LIN {X 0,Y 418.244,Z 286.013,A -85,B 0,C 180,E1 -10136.324,E2 -10136.324} C_VEL
LIN {X 0,Y 418.278,Z 286.189,A -85,B 0,C 180,E1 -10136.962,E2 -10136.962} C_VEL
LIN {X 0,Y 422.235,Z 301.677,A -85,B 0,C 180,E1 -10140.044,E2 -10140.044} C_VEL
LIN {X 0,Y 424.407,Z 311.611,A -85,B 0,C 180,E1 -10141.923,E2 -10141.923} C_VEL
LIN {X 0,Y 424.445,Z 314.254,A -85,B 0,C 180,E1 -10142.379,E2 -10142.379} C_VEL
LIN {X 0,Y 424.103,Z 317.879,A -85,B 0,C 180,E1 -10142.98,E2 -10142.98} C_VEL
LIN {X 0,Y 430.223,Z 348.762,A -85,B 0,C 180,E1 -10143.957,E2 -10143.957} C_VEL
LIN {X 0,Y 430.634,Z 351.197,A -85,B 0,C 180,E1 -10144.027,E2 -10144.027} C_VEL
LIN {X 0,Y 428.256,Z 483.679,A -85,B 0,C 180,E1 -10146.294,E2 -10146.294} C_VEL
LIN {X 0,Y 427.572,Z 499.207,A -85,B 0,C 180,E1 -10146.735,E2 -10146.735} C_VEL
LIN {X 0,Y 426.692,Z 513.897,A -85,B 0,C 180,E1 -10147.343,E2 -10147.343} C_VEL
LIN {X 0,Y 425.714,Z 527.179,A -85,B 0,C 180,E1 -10148.068,E2 -10148.068} C_VEL
LIN {X 0,Y 424.501,Z 541.084,A -85,B 0,C 180,E1 -10149.022,E2 -10149.022} C_VEL
LIN {X 0,Y 423.263,Z 553.827,A -85,B 0,C 180,E1 -10150.1,E2 -10150.1} C_VEL
LIN {X 0,Y 421.996,Z 566.72,A -85,B 0,C 180,E1 -10151.428,E2 -10151.428} C_VEL
LIN {X 0,Y 420.886,Z 577.517,A -85,B 0,C 180,E1 -10152.76,E2 -10152.76} C_VEL
LIN {X 0,Y 419.829,Z 587.51,A -85,B 0,C 180,E1 -10154.216,E2 -10154.216} C_VEL
LIN {X 0,Y 418.872,Z 597.29,A -85,B 0,C 180,E1 -10155.92,E2 -10155.92} C_VEL
LIN {X 0,Y 418.217,Z 605.457,A -85,B 0,C 180,E1 -10157.628,E2 -10157.628} C_VEL
LIN {X 0,Y 417.695,Z 612.208,A -85,B 0,C 180,E1 -10159.334,E2 -10159.334} C_VEL
LIN {X 0,Y 417.31,Z 618.446,A -85,B 0,C 180,E1 -10161.282,E2 -10161.282} C_VEL
LIN {X 0,Y 417.147,Z 623.274,A -85,B 0,C 180,E1 -10163.227,E2 -10163.227} C_VEL
LIN {X 0,Y 417.046,Z 626.811,A -85,B 0,C 180,E1 -10165.167,E2 -10165.167} C_VEL
LIN {X 0,Y 417.01,Z 629.139,A -85,B 0,C 180,E1 -10167.102,E2 -10167.102} C_VEL
LIN {X 0,Y 417.008,Z 630.31,A -85,B 0,C 180,E1 -10169.034,E2 -10169.034} C_VEL
LIN {X 0,Y 417.008,Z 630.308,A -85,B 0,C 180,E1 -10170.966,E2 -10170.966} C_VEL
LIN {X 0,Y 417.01,Z 629.131,A -85,B 0,C 180,E1 -10172.898,E2 -10172.898} C_VEL
LIN {X 0,Y 417.025,Z 626.8,A -85,B 0,C 180,E1 -10174.834,E2 -10174.834} C_VEL
LIN {X 0,Y 417.139,Z 623.267,A -85,B 0,C 180,E1 -10176.773,E2 -10176.773} C_VEL
LIN {X 0,Y 417.31,Z 618.438,A -85,B 0,C 180,E1 -10178.718,E2 -10178.718} C_VEL
LIN {X 0,Y 417.694,Z 612.188,A -85,B 0,C 180,E1 -10180.666,E2 -10180.666} C_VEL
LIN {X 0,Y 418.223,Z 605.432,A -85,B 0,C 180,E1 -10182.372,E2 -10182.372} C_VEL
LIN {X 0,Y 419.012,Z 596.002,A -85,B 0,C 180,E1 -10184.323,E2 -10184.323} C_VEL
LIN {X 0,Y 419.969,Z 585.957,A -85,B 0,C 180,E1 -10186.028,E2 -10186.028} C_VEL
LIN {X 0,Y 421.237,Z 574.541,A -85,B 0,C 180,E1 -10187.629,E2 -10187.629} C_VEL
LIN {X 0,Y 422.391,Z 562.305,A -85,B 0,C 180,E1 -10189.058,E2 -10189.058} C_VEL
LIN {X 0,Y 423.709,Z 549.847,A -85,B 0,C 180,E1 -10190.258,E2 -10190.258} C_VEL
LIN {X 0,Y 424.949,Z 536.202,A -85,B 0,C 180,E1 -10191.336,E2 -10191.336} C_VEL
LIN {X 0,Y 426.1,Z 522.072,A -85,B 0,C 180,E1 -10192.229,E2 -10192.229} C_VEL
LIN {X 0,Y 427.157,Z 506.655,A -85,B 0,C 180,E1 -10192.975,E2 -10192.975} C_VEL
LIN {X 0,Y 427.948,Z 491.612,A -85,B 0,C 180,E1 -10193.5,E2 -10193.5} C_VEL
LIN {X 0,Y 428.422,Z 475.672,A -85,B 0,C 180,E1 -10193.857,E2 -10193.857} C_VEL
LIN {X 0,Y 430.58,Z 352.154,A -85,B 0,C 180,E1 -10195.952,E2 -10195.952} C_VEL
LIN {X 0,Y 429.942,Z 347.275,A -85,B 0,C 180,E1 -10196.081,E2 -10196.081} C_VEL
LIN {X 0,Y 424.097,Z 317.761,A -85,B 0,C 180,E1 -10197.032,E2 -10197.032} C_VEL
LIN {X 0,Y 424.547,Z 312.878,A -85,B 0,C 180,E1 -10197.841,E2 -10197.841} C_VEL
LIN {X 0,Y 422.7,Z 303.593,A -85,B 0,C 180,E1 -10199.576,E2 -10199.576} C_VEL
LIN {X 0,Y 419.42,Z 290.486,A -85,B 0,C 180,E1 -10202.152,E2 -10202.152} C_VEL
LIN {X 0,Y 418.237,Z 286.011,A -85,B 0,C 180,E1 -10203.1,E2 -10203.1} C_VEL
LIN {X 0,Y 418.236,Z 286.014,A -85,B 0,C 180,E1 -10206.236,E2 -10206.236} C_VEL
LIN {X 0,Y 418.192,Z 286.02,A -85,B 0,C 180,E1 -10209.687,E2 -10209.687} C_VEL
LIN {X 0,Y 418.202,Z 286.02,A -85,B 0,C 180,E1 -10212.317,E2 -10212.317} C_VEL
LIN {X 0,Y 418.227,Z 286.013,A -85,B 0,C 180,E1 -10215.108,E2 -10215.108} C_VEL
LIN {X 0,Y 418.215,Z 286.016,A -85,B 0,C 180,E1 -10217.764,E2 -10217.764} C_VEL
LIN {X 0,Y 418.225,Z 286.015,A -85,B 0,C 180,E1 -10221.555,E2 -10221.555} C_VEL
LIN {X 0,Y 418.24,Z 286.008,A -85,B 0,C 180,E1 -10225.157,E2 -10225.157} C_VEL
LIN {X 0,Y 418.233,Z 286.01,A -85,B 0,C 180,E1 -10227.471,E2 -10227.471} C_VEL
LIN {X 0,Y 418.252,Z 286.007,A -85,B 0,C 180,E1 -10230.897,E2 -10230.897} C_VEL
LIN {X 0,Y 418.207,Z 286.017,A -85,B 0,C 180,E1 -10234.092,E2 -10234.092} C_VEL
LIN {X 0,Y 418.216,Z 286.014,A -85,B 0,C 180,E1 -10237.263,E2 -10237.263} C_VEL
LIN {X 0,Y 418.272,Z 285.991,A -85,B 0,C 180,E1 -10240.364,E2 -10240.364} C_VEL
LIN {X 0,Y 418.304,Z 286,A -85,B 0,C 180,E1 -10243.404,E2 -10243.404} C_VEL
LIN {X 0,Y 418.334,Z 285.993,A -85,B 0,C 180,E1 -10247,E2 -10247} C_VEL
LIN {X 0,Y 418.306,Z 285.996,A -85,B 0,C 180,E1 -10250.328,E2 -10250.328} C_VEL
LIN {X 0,Y 418.448,Z 285.988,A -85,B 0,C 180,E1 -10253.248,E2 -10253.248} C_VEL
LIN {X 0,Y 418.307,Z 285.999,A -85,B 0,C 180,E1 -10255.181,E2 -10255.181} C_VEL
LIN {X 0,Y 418.52,Z 285.97,A -85,B 0,C 180,E1 -10258.075,E2 -10258.075} C_VEL
LIN {X 0,Y 418.394,Z 285.993,A -85,B 0,C 180,E1 -10260.963,E2 -10260.963} C_VEL
LIN {X 0,Y 418.469,Z 285.978,A -85,B 0,C 180,E1 -10262.888,E2 -10262.888} C_VEL
LIN {X 0,Y 418.452,Z 285.98,A -85,B 0,C 180,E1 -10266.593,E2 -10266.593} C_VEL
LIN {X 0,Y 418.324,Z 285.999,A -85,B 0,C 180,E1 -10269.672,E2 -10269.672} C_VEL
LIN {X 0,Y 418.335,Z 286.002,A -85,B 0,C 180,E1 -10273.001,E2 -10273.001} C_VEL
LIN {X 0,Y 418.301,Z 286.004,A -85,B 0,C 180,E1 -10276.735,E2 -10276.735} C_VEL
LIN {X 0,Y 418.259,Z 285.992,A -85,B 0,C 180,E1 -10279.79,E2 -10279.79} C_VEL
LIN {X 0,Y 418.227,Z 286.008,A -85,B 0,C 180,E1 -10282.737,E2 -10282.737} C_VEL
LIN {X 0,Y 418.251,Z 286.002,A -85,B 0,C 180,E1 -10285.905,E2 -10285.905} C_VEL
LIN {X 0,Y 418.26,Z 286.005,A -85,B 0,C 180,E1 -10289.105,E2 -10289.105} C_VEL
LIN {X 0,Y 418.234,Z 286.009,A -85,B 0,C 180,E1 -10292.529,E2 -10292.529} C_VEL
LIN {X 0,Y 418.234,Z 286.01,A -85,B 0,C 180,E1 -10296.025,E2 -10296.025} C_VEL
LIN {X 0,Y 418.238,Z 286.007,A -85,B 0,C 180,E1 -10299.684,E2 -10299.684} C_VEL
LIN {X 0,Y 418.223,Z 286.013,A -85,B 0,C 180,E1 -10302.322,E2 -10302.322} C_VEL
LIN {X 0,Y 418.23,Z 286.015,A -85,B 0,C 180,E1 -10305.11,E2 -10305.11} C_VEL
LIN {X 0,Y 418.235,Z 286.012,A -85,B 0,C 180,E1 -10307.768,E2 -10307.768} C_VEL
LIN {X 0,Y 418.254,Z 286.007,A -85,B 0,C 180,E1 -10310.619,E2 -10310.619} C_VEL
LIN {X 0,Y 418.239,Z 286.008,A -85,B 0,C 180,E1 -10313.977,E2 -10313.977} C_VEL
LIN {X 0,Y 418.254,Z 286.009,A -85,B 0,C 180,E1 -10317.157,E2 -10317.157} C_VEL
LIN {X 0,Y 418.268,Z 286.038,A -85,B 0,C 180,E1 -10320.426,E2 -10320.426} C_VEL
LIN {X 0,Y 421.092,Z 297.257,A -85,B 0,C 180,E1 -10322.844,E2 -10322.844} C_VEL
LIN {X 0,Y 429.309,Z 316.827,A -85,B 0,C 180,E1 -10323.769,E2 -10323.769} C_VEL
LIN {X 0,Y 430.945,Z 324.515,A -85,B 0,C 180,E1 -10324.017,E2 -10324.017} C_VEL
LIN {X 0,Y 428.589,Z 458.839,A -85,B 0,C 180,E1 -10326.313,E2 -10326.313} C_VEL
LIN {X 0,Y 428.076,Z 473.456,A -85,B 0,C 180,E1 -10326.7,E2 -10326.7} C_VEL
LIN {X 0,Y 427.345,Z 488.698,A -85,B 0,C 180,E1 -10327.299,E2 -10327.299} C_VEL
LIN {X 0,Y 426.339,Z 503.778,A -85,B 0,C 180,E1 -10328.102,E2 -10328.102} C_VEL
LIN {X 0,Y 425.211,Z 517.76,A -85,B 0,C 180,E1 -10329.059,E2 -10329.059} C_VEL
LIN {X 0,Y 423.983,Z 530.538,A -85,B 0,C 180,E1 -10330.135,E2 -10330.135} C_VEL
LIN {X 0,Y 422.724,Z 543.427,A -85,B 0,C 180,E1 -10331.464,E2 -10331.464} C_VEL
LIN {X 0,Y 421.603,Z 554.154,A -85,B 0,C 180,E1 -10332.79,E2 -10332.79} C_VEL
LIN {X 0,Y 421.269,Z 557.507,A -85,B 0,C 180,E1 -10333.249,E2 -10333.249} C_VEL
LIN {X 0,Y 420.236,Z 561.612,A -85,B 0,C 180,E1 -10333.811,E2 -10333.811} C_VEL
LIN {X 0,Y 416.771,Z 568.053,A -85,B 0,C 180,E1 -10334.729,E2 -10334.729} C_VEL
LIN {X 0,Y 413.273,Z 574.004,A -85,B 0,C 180,E1 -10335.715,E2 -10335.715} C_VEL
LIN {X 0,Y 412.208,Z 577.344,A -85,B 0,C 180,E1 -10336.377,E2 -10336.377} C_VEL
LIN {X 0,Y 411.56,Z 585.076,A -85,B 0,C 180,E1 -10338.176,E2 -10338.176} C_VEL
LIN {X 0,Y 410.84,Z 592.015,A -85,B 0,C 180,E1 -10340.151,E2 -10340.151} C_VEL
LIN {X 0,Y 410.445,Z 597.464,A -85,B 0,C 180,E1 -10342.127,E2 -10342.127} C_VEL
LIN {X 0,Y 410.194,Z 601.578,A -85,B 0,C 180,E1 -10344.1,E2 -10344.1} C_VEL
LIN {X 0,Y 409.99,Z 604.471,A -85,B 0,C 180,E1 -10346.068,E2 -10346.068} C_VEL
LIN {X 0,Y 410.008,Z 606.209,A -85,B 0,C 180,E1 -10348.035,E2 -10348.035} C_VEL
LIN {X 0,Y 409.925,Z 606.819,A -85,B 0,C 180,E1 -10350,E2 -10350} C_VEL
LIN {X 0,Y 410.008,Z 606.257,A -85,B 0,C 180,E1 -10351.965,E2 -10351.965} C_VEL
LIN {X 0,Y 409.98,Z 604.584,A -85,B 0,C 180,E1 -10353.932,E2 -10353.932} C_VEL
LIN {X 0,Y 410.182,Z 601.751,A -85,B 0,C 180,E1 -10355.9,E2 -10355.9} C_VEL
LIN {X 0,Y 410.411,Z 597.698,A -85,B 0,C 180,E1 -10357.874,E2 -10357.874} C_VEL
LIN {X 0,Y 410.824,Z 592.321,A -85,B 0,C 180,E1 -10359.85,E2 -10359.85} C_VEL
LIN {X 0,Y 411.541,Z 585.465,A -85,B 0,C 180,E1 -10361.825,E2 -10361.825} C_VEL
LIN {X 0,Y 412.292,Z 576.91,A -85,B 0,C 180,E1 -10363.806,E2 -10363.806} C_VEL
LIN {X 0,Y 413.318,Z 567.808,A -85,B 0,C 180,E1 -10365.534,E2 -10365.534} C_VEL
LIN {X 0,Y 414.347,Z 558.53,A -85,B 0,C 180,E1 -10367.012,E2 -10367.012} C_VEL
LIN {X 0,Y 415.663,Z 546.61,A -85,B 0,C 180,E1 -10368.6,E2 -10368.6} C_VEL
LIN {X 0,Y 416.981,Z 534.265,A -85,B 0,C 180,E1 -10369.956,E2 -10369.956} C_VEL
LIN {X 0,Y 418.37,Z 520.731,A -85,B 0,C 180,E1 -10371.171,E2 -10371.171} C_VEL
LIN {X 0,Y 419.534,Z 507.419,A -85,B 0,C 180,E1 -10372.142,E2 -10372.142} C_VEL
LIN {X 0,Y 420.633,Z 492.721,A -85,B 0,C 180,E1 -10372.988,E2 -10372.988} C_VEL
LIN {X 0,Y 421.422,Z 478.095,A -85,B 0,C 180,E1 -10373.625,E2 -10373.625} C_VEL
LIN {X 0,Y 422.01,Z 463.194,A -85,B 0,C 180,E1 -10374.079,E2 -10374.079} C_VEL
LIN {X 0,Y 422.988,Z 418.773,A -85,B 0,C 180,E1 -10374.87,E2 -10374.87} C_VEL
LIN {X 0,Y 424.551,Z 324.982,A -85,B 0,C 180,E1 -10376.498,E2 -10376.498} C_VEL
LIN {X 0,Y 422.627,Z 317.569,A -85,B 0,C 180,E1 -10376.767,E2 -10376.767} C_VEL
LIN {X 0,Y 413.797,Z 297.173,A -85,B 0,C 180,E1 -10377.792,E2 -10377.792} C_VEL
LIN {X 0,Y 411.215,Z 286.891,A -85,B 0,C 180,E1 -10380.134,E2 -10380.134} C_VEL
LIN {X 0,Y 411.204,Z 286.894,A -85,B 0,C 180,E1 -10383.155,E2 -10383.155} C_VEL
LIN {X 0,Y 411.191,Z 286.894,A -85,B 0,C 180,E1 -10386.552,E2 -10386.552} C_VEL
LIN {X 0,Y 411.208,Z 286.884,A -85,B 0,C 180,E1 -10389.727,E2 -10389.727} C_VEL
LIN {X 0,Y 411.168,Z 286.894,A -85,B 0,C 180,E1 -10393.133,E2 -10393.133} C_VEL
LIN {X 0,Y 411.161,Z 286.893,A -85,B 0,C 180,E1 -10395.88,E2 -10395.88} C_VEL
LIN {X 0,Y 411.154,Z 286.882,A -85,B 0,C 180,E1 -10398.771,E2 -10398.771} C_VEL
LIN {X 0,Y 411.182,Z 286.884,A -85,B 0,C 180,E1 -10402.025,E2 -10402.025} C_VEL
LIN {X 0,Y 411.185,Z 286.891,A -85,B 0,C 180,E1 -10405.664,E2 -10405.664} C_VEL
LIN {X 0,Y 411.18,Z 286.875,A -85,B 0,C 180,E1 -10409.151,E2 -10409.151} C_VEL
LIN {X 0,Y 411.258,Z 286.882,A -85,B 0,C 180,E1 -10412.698,E2 -10412.698} C_VEL
LIN {X 0,Y 411.201,Z 286.887,A -85,B 0,C 180,E1 -10415.783,E2 -10415.783} C_VEL
LIN {X 0,Y 411.186,Z 286.889,A -85,B 0,C 180,E1 -10418.965,E2 -10418.965} C_VEL
LIN {X 0,Y 411.234,Z 286.878,A -85,B 0,C 180,E1 -10422.084,E2 -10422.084} C_VEL
LIN {X 0,Y 411.247,Z 286.882,A -85,B 0,C 180,E1 -10425.147,E2 -10425.147} C_VEL
LIN {X 0,Y 411.27,Z 286.877,A -85,B 0,C 180,E1 -10428.167,E2 -10428.167} C_VEL
LIN {X 0,Y 411.427,Z 286.856,A -85,B 0,C 180,E1 -10432.191,E2 -10432.191} C_VEL
LIN {X 0,Y 411.432,Z 286.858,A -85,B 0,C 180,E1 -10434.117,E2 -10434.117} C_VEL
LIN {X 0,Y 411.497,Z 286.85,A -85,B 0,C 180,E1 -10438.042,E2 -10438.042} C_VEL
LIN {X 0,Y 411.622,Z 286.83,A -85,B 0,C 180,E1 -10440,E2 -10440} C_VEL
LIN {X 0,Y 411.421,Z 286.86,A -85,B 0,C 180,E1 -10442.937,E2 -10442.937} C_VEL
LIN {X 0,Y 411.419,Z 286.863,A -85,B 0,C 180,E1 -10446.868,E2 -10446.868} C_VEL
LIN {X 0,Y 411.27,Z 286.874,A -85,B 0,C 180,E1 -10449.839,E2 -10449.839} C_VEL
LIN {X 0,Y 411.294,Z 286.87,A -85,B 0,C 180,E1 -10453.104,E2 -10453.104} C_VEL
LIN {X 0,Y 411.247,Z 286.88,A -85,B 0,C 180,E1 -10456.889,E2 -10456.889} C_VEL
LIN {X 0,Y 411.22,Z 286.888,A -85,B 0,C 180,E1 -10459.987,E2 -10459.987} C_VEL
LIN {X 0,Y 411.176,Z 286.891,A -85,B 0,C 180,E1 -10463.149,E2 -10463.149} C_VEL
LIN {X 0,Y 411.164,Z 286.892,A -85,B 0,C 180,E1 -10466.386,E2 -10466.386} C_VEL
LIN {X 0,Y 411.188,Z 286.89,A -85,B 0,C 180,E1 -10469.714,E2 -10469.714} C_VEL
LIN {X 0,Y 411.195,Z 286.882,A -85,B 0,C 180,E1 -10473.157,E2 -10473.157} C_VEL
LIN {X 0,Y 411.179,Z 286.889,A -85,B 0,C 180,E1 -10476.552,E2 -10476.552} C_VEL
LIN {X 0,Y 411.159,Z 286.884,A -85,B 0,C 180,E1 -10479.721,E2 -10479.721} C_VEL
LIN {X 0,Y 411.157,Z 286.893,A -85,B 0,C 180,E1 -10483.136,E2 -10483.136} C_VEL
LIN {X 0,Y 411.156,Z 286.896,A -85,B 0,C 180,E1 -10485.883,E2 -10485.883} C_VEL
LIN {X 0,Y 411.14,Z 286.895,A -85,B 0,C 180,E1 -10488.775,E2 -10488.775} C_VEL
LIN {X 0,Y 411.176,Z 286.892,A -85,B 0,C 180,E1 -10492.026,E2 -10492.026} C_VEL
LIN {X 0,Y 411.201,Z 286.89,A -85,B 0,C 180,E1 -10495.667,E2 -10495.667} C_VEL
LIN {X 0,Y 411.228,Z 287.031,A -85,B 0,C 180,E1 -10496.518,E2 -10496.518} C_VEL
LIN {X 0,Y 415.224,Z 302.546,A -85,B 0,C 180,E1 -10499.679,E2 -10499.679} C_VEL
LIN {X 0,Y 417.696,Z 314.046,A -85,B 0,C 180,E1 -10501.894,E2 -10501.894} C_VEL
LIN {X 0,Y 417.508,Z 317.887,A -85,B 0,C 180,E1 -10502.524,E2 -10502.524} C_VEL
LIN {X 0,Y 423.554,Z 348.293,A -85,B 0,C 180,E1 -10503.51,E2 -10503.51} C_VEL
LIN {X 0,Y 424.204,Z 351.82,A -85,B 0,C 180,E1 -10503.619,E2 -10503.619} C_VEL
LIN {X 0,Y 421.839,Z 481.988,A -85,B 0,C 180,E1 -10505.878,E2 -10505.878} C_VEL
LIN {X 0,Y 421.199,Z 497.183,A -85,B 0,C 180,E1 -10506.296,E2 -10506.296} C_VEL
LIN {X 0,Y 420.276,Z 511.874,A -85,B 0,C 180,E1 -10506.886,E2 -10506.886} C_VEL
LIN {X 0,Y 419.259,Z 524.987,A -85,B 0,C 180,E1 -10507.583,E2 -10507.583} C_VEL
LIN {X 0,Y 417.986,Z 539.298,A -85,B 0,C 180,E1 -10508.55,E2 -10508.55} C_VEL
LIN {X 0,Y 416.671,Z 552.33,A -85,B 0,C 180,E1 -10509.643,E2 -10509.643} C_VEL
LIN {X 0,Y 415.395,Z 564.368,A -85,B 0,C 180,E1 -10510.865,E2 -10510.865} C_VEL
LIN {X 0,Y 414.275,Z 575.524,A -85,B 0,C 180,E1 -10512.221,E2 -10512.221} C_VEL
LIN {X 0,Y 413.049,Z 585.786,A -85,B 0,C 180,E1 -10513.696,E2 -10513.696} C_VEL
LIN {X 0,Y 412.058,Z 595.825,A -85,B 0,C 180,E1 -10515.43,E2 -10515.43} C_VEL
LIN {X 0,Y 411.262,Z 604.165,A -85,B 0,C 180,E1 -10517.165,E2 -10517.165} C_VEL
LIN {X 0,Y 410.853,Z 610.183,A -85,B 0,C 180,E1 -10518.655,E2 -10518.655} C_VEL
LIN {X 0,Y 410.32,Z 616.806,A -85,B 0,C 180,E1 -10520.636,E2 -10520.636} C_VEL
LIN {X 0,Y 410.107,Z 621.994,A -85,B 0,C 180,E1 -10522.616,E2 -10522.616} C_VEL
LIN {X 0,Y 409.975,Z 624.995,A -85,B 0,C 180,E1 -10524.097,E2 -10524.097} C_VEL
LIN {X 0,Y 409.893,Z 627.918,A -85,B 0,C 180,E1 -10526.067,E2 -10526.067} C_VEL
LIN {X 0,Y 409.961,Z 629.665,A -85,B 0,C 180,E1 -10528.035,E2 -10528.035} C_VEL
LIN {X 0,Y 409.923,Z 630.262,A -85,B 0,C 180,E1 -10530,E2 -10530} C_VEL
LIN {X 0,Y 409.961,Z 629.661,A -85,B 0,C 180,E1 -10531.965,E2 -10531.965} C_VEL
LIN {X 0,Y 409.89,Z 627.908,A -85,B 0,C 180,E1 -10533.933,E2 -10533.933} C_VEL
LIN {X 0,Y 409.975,Z 624.984,A -85,B 0,C 180,E1 -10535.903,E2 -10535.903} C_VEL
LIN {X 0,Y 410.131,Z 620.816,A -85,B 0,C 180,E1 -10537.879,E2 -10537.879} C_VEL
LIN {X 0,Y 410.379,Z 615.293,A -85,B 0,C 180,E1 -10539.861,E2 -10539.861} C_VEL
LIN {X 0,Y 410.991,Z 608.274,A -85,B 0,C 180,E1 -10541.841,E2 -10541.841} C_VEL
LIN {X 0,Y 411.588,Z 600.675,A -85,B 0,C 180,E1 -10543.597,E2 -10543.597} C_VEL
LIN {X 0,Y 412.489,Z 591.709,A -85,B 0,C 180,E1 -10545.312,E2 -10545.312} C_VEL
LIN {X 0,Y 413.472,Z 582.478,A -85,B 0,C 180,E1 -10546.795,E2 -10546.795} C_VEL
LIN {X 0,Y 414.563,Z 572.303,A -85,B 0,C 180,E1 -10548.186,E2 -10548.186} C_VEL
LIN {X 0,Y 415.856,Z 559.74,A -85,B 0,C 180,E1 -10549.626,E2 -10549.626} C_VEL
LIN {X 0,Y 417.28,Z 546.775,A -85,B 0,C 180,E1 -10550.842,E2 -10550.842} C_VEL
LIN {X 0,Y 418.526,Z 534.225,A -85,B 0,C 180,E1 -10551.809,E2 -10551.809} C_VEL
LIN {X 0,Y 419.621,Z 520.739,A -85,B 0,C 180,E1 -10552.656,E2 -10552.656} C_VEL
LIN {X 0,Y 420.639,Z 505.747,A -85,B 0,C 180,E1 -10553.382,E2 -10553.382} C_VEL
LIN {X 0,Y 421.442,Z 491.397,A -85,B 0,C 180,E1 -10553.885,E2 -10553.885} C_VEL
LIN {X 0,Y 421.948,Z 475.45,A -85,B 0,C 180,E1 -10554.247,E2 -10554.247} C_VEL
LIN {X 0,Y 424.196,Z 352.499,A -85,B 0,C 180,E1 -10556.362,E2 -10556.362} C_VEL
LIN {X 0,Y 419.4,Z 326.937,A -85,B 0,C 180,E1 -10557.164,E2 -10557.164} C_VEL
LIN {X 0,Y 417.45,Z 317.556,A -85,B 0,C 180,E1 -10557.497,E2 -10557.497} C_VEL
LIN {X 0,Y 417.685,Z 313.984,A -85,B 0,C 180,E1 -10558.107,E2 -10558.107} C_VEL
LIN {X 0,Y 415.482,Z 303.69,A -85,B 0,C 180,E1 -10560.085,E2 -10560.085} C_VEL
LIN {X 0,Y 412.102,Z 290.329,A -85,B 0,C 180,E1 -10562.782,E2 -10562.782} C_VEL
LIN {X 0,Y 411.21,Z 286.888,A -85,B 0,C 180,E1 -10563.52,E2 -10563.52} C_VEL
LIN {X 0,Y 411.181,Z 286.892,A -85,B 0,C 180,E1 -10566.742,E2 -10566.742} C_VEL
LIN {X 0,Y 411.161,Z 286.895,A -85,B 0,C 180,E1 -10569.719,E2 -10569.719} C_VEL
LIN {X 0,Y 411.156,Z 286.894,A -85,B 0,C 180,E1 -10573.134,E2 -10573.134} C_VEL
LIN {X 0,Y 411.157,Z 286.897,A -85,B 0,C 180,E1 -10575.881,E2 -10575.881} C_VEL
LIN {X 0,Y 411.141,Z 286.895,A -85,B 0,C 180,E1 -10578.773,E2 -10578.773} C_VEL
LIN {X 0,Y 411.172,Z 286.892,A -85,B 0,C 180,E1 -10582.024,E2 -10582.024} C_VEL
LIN {X 0,Y 411.192,Z 286.886,A -85,B 0,C 180,E1 -10585.123,E2 -10585.123} C_VEL
LIN {X 0,Y 411.154,Z 286.896,A -85,B 0,C 180,E1 -10588.002,E2 -10588.002} C_VEL
LIN {X 0,Y 411.169,Z 286.893,A -85,B 0,C 180,E1 -10591.406,E2 -10591.406} C_VEL
LIN {X 0,Y 411.177,Z 286.89,A -85,B 0,C 180,E1 -10594.941,E2 -10594.941} C_VEL
LIN {X 0,Y 411.192,Z 286.89,A -85,B 0,C 180,E1 -10597.913,E2 -10597.913} C_VEL
LIN {X 0,Y 411.206,Z 286.869,A -85,B 0,C 180,E1 -10601.051,E2 -10601.051} C_VEL
LIN {X 0,Y 411.24,Z 286.883,A -85,B 0,C 180,E1 -10604.131,E2 -10604.131} C_VEL
LIN {X 0,Y 411.29,Z 286.866,A -85,B 0,C 180,E1 -10607.165,E2 -10607.165} C_VEL
LIN {X 0,Y 411.26,Z 286.874,A -85,B 0,C 180,E1 -10610.161,E2 -10610.161} C_VEL
LIN {X 0,Y 411.413,Z 286.863,A -85,B 0,C 180,E1 -10613.132,E2 -10613.132} C_VEL
LIN {X 0,Y 411.279,Z 286.874,A -85,B 0,C 180,E1 -10615.099,E2 -10615.099} C_VEL
LIN {X 0,Y 411.49,Z 286.846,A -85,B 0,C 180,E1 -10618.043,E2 -10618.043} C_VEL
LIN {X 0,Y 411.494,Z 286.847,A -85,B 0,C 180,E1 -10621.958,E2 -10621.958} C_VEL
LIN {X 0,Y 411.412,Z 286.857,A -85,B 0,C 180,E1 -10626.596,E2 -10626.596} C_VEL
LIN {X 0,Y 411.306,Z 286.875,A -85,B 0,C 180,E1 -10628.846,E2 -10628.846} C_VEL
LIN {X 0,Y 411.27,Z 286.878,A -85,B 0,C 180,E1 -10631.833,E2 -10631.833} C_VEL
LIN {X 0,Y 411.245,Z 286.881,A -85,B 0,C 180,E1 -10634.853,E2 -10634.853} C_VEL
LIN {X 0,Y 411.234,Z 286.88,A -85,B 0,C 180,E1 -10637.916,E2 -10637.916} C_VEL
LIN {X 0,Y 411.186,Z 286.872,A -85,B 0,C 180,E1 -10641.035,E2 -10641.035} C_VEL
LIN {X 0,Y 411.207,Z 286.886,A -85,B 0,C 180,E1 -10644.217,E2 -10644.217} C_VEL
LIN {X 0,Y 411.25,Z 286.867,A -85,B 0,C 180,E1 -10647.478,E2 -10647.478} C_VEL
LIN {X 0,Y 411.181,Z 286.894,A -85,B 0,C 180,E1 -10650.848,E2 -10650.848} C_VEL
LIN {X 0,Y 411.184,Z 286.889,A -85,B 0,C 180,E1 -10654.336,E2 -10654.336} C_VEL
LIN {X 0,Y 411.185,Z 286.886,A -85,B 0,C 180,E1 -10657.975,E2 -10657.975} C_VEL
LIN {X 0,Y 411.157,Z 286.894,A -85,B 0,C 180,E1 -10661.229,E2 -10661.229} C_VEL
LIN {X 0,Y 411.17,Z 286.893,A -85,B 0,C 180,E1 -10664.491,E2 -10664.491} C_VEL
LIN {X 0,Y 411.173,Z 286.893,A -85,B 0,C 180,E1 -10668.196,E2 -10668.196} C_VEL
LIN {X 0,Y 411.218,Z 286.882,A -85,B 0,C 180,E1 -10670.777,E2 -10670.777} C_VEL
LIN {X 0,Y 411.194,Z 286.885,A -85,B 0,C 180,E1 -10674.472,E2 -10674.472} C_VEL
LIN {X 0,Y 411.205,Z 286.886,A -85,B 0,C 180,E1 -10676.874,E2 -10676.874} C_VEL
LIN {X 0,Y 411.221,Z 286.926,A -85,B 0,C 180,E1 -10680.008,E2 -10680.008} C_VEL
LIN {X 0,Y 413.864,Z 297.254,A -85,B 0,C 180,E1 -10682.324,E2 -10682.324} C_VEL
LIN {X 0,Y 423.139,Z 318.948,A -85,B 0,C 180,E1 -10683.392,E2 -10683.392} C_VEL
LIN {X 0,Y 424.531,Z 325.264,A -85,B 0,C 180,E1 -10683.604,E2 -10683.604} C_VEL
LIN {X 0,Y 422.503,Z 438.469,A -85,B 0,C 180,E1 -10685.559,E2 -10685.559} C_VEL
LIN {X 0,Y 421.964,Z 463.218,A -85,B 0,C 180,E1 -10686.016,E2 -10686.016} C_VEL
LIN {X 0,Y 421.361,Z 478.668,A -85,B 0,C 180,E1 -10686.492,E2 -10686.492} C_VEL
LIN {X 0,Y 420.666,Z 492.476,A -85,B 0,C 180,E1 -10687.098,E2 -10687.098} C_VEL
LIN {X 0,Y 419.612,Z 505.967,A -85,B 0,C 180,E1 -10687.862,E2 -10687.862} C_VEL
LIN {X 0,Y 418.432,Z 519.546,A -85,B 0,C 180,E1 -10688.832,E2 -10688.832} C_VEL
LIN {X 0,Y 417.062,Z 533.318,A -85,B 0,C 180,E1 -10690.048,E2 -10690.048} C_VEL
LIN {X 0,Y 415.783,Z 545.736,A -85,B 0,C 180,E1 -10691.395,E2 -10691.395} C_VEL
LIN {X 0,Y 414.61,Z 556.132,A -85,B 0,C 180,E1 -10692.745,E2 -10692.745} C_VEL
LIN {X 0,Y 413.525,Z 565.772,A -85,B 0,C 180,E1 -10694.222,E2 -10694.222} C_VEL
LIN {X 0,Y 412.462,Z 575.219,A -85,B 0,C 180,E1 -10695.948,E2 -10695.948} C_VEL
LIN {X 0,Y 412.208,Z 577.344,A -85,B 0,C 180,E1 -10696.377,E2 -10696.377} C_VEL
LIN {X 0,Y 411.188,Z 580.565,A -85,B 0,C 180,E1 -10697.056,E2 -10697.056} C_VEL
LIN {X 0,Y 407.883,Z 585.558,A -85,B 0,C 180,E1 -10698.162,E2 -10698.162} C_VEL
LIN {X 0,Y 404.661,Z 590.076,A -85,B 0,C 180,E1 -10699.321,E2 -10699.321} C_VEL
LIN {X 0,Y 403.782,Z 592.508,A -85,B 0,C 180,E1 -10700.074,E2 -10700.074} C_VEL
LIN {X 0,Y 403.391,Z 597.669,A -85,B 0,C 180,E1 -10701.988,E2 -10701.988} C_VEL
LIN {X 0,Y 403.117,Z 601.782,A -85,B 0,C 180,E1 -10703.996,E2 -10703.996} C_VEL
LIN {X 0,Y 402.909,Z 604.675,A -85,B 0,C 180,E1 -10705.999,E2 -10705.999} C_VEL
LIN {X 0,Y 402.921,Z 606.412,A -85,B 0,C 180,E1 -10708.001,E2 -10708.001} C_VEL
LIN {X 0,Y 402.85,Z 607.022,A -85,B 0,C 180,E1 -10710,E2 -10710} C_VEL
LIN {X 0,Y 402.921,Z 606.46,A -85,B 0,C 180,E1 -10711.999,E2 -10711.999} C_VEL
LIN {X 0,Y 402.9,Z 604.786,A -85,B 0,C 180,E1 -10714.001,E2 -10714.001} C_VEL
LIN {X 0,Y 403.106,Z 601.954,A -85,B 0,C 180,E1 -10716.004,E2 -10716.004} C_VEL
LIN {X 0,Y 403.367,Z 597.9,A -85,B 0,C 180,E1 -10718.012,E2 -10718.012} C_VEL
LIN {X 0,Y 403.793,Z 592.524,A -85,B 0,C 180,E1 -10720.023,E2 -10720.023} C_VEL
LIN {X 0,Y 404.558,Z 585.667,A -85,B 0,C 180,E1 -10722.032,E2 -10722.032} C_VEL
LIN {X 0,Y 405.386,Z 577.111,A -85,B 0,C 180,E1 -10724.046,E2 -10724.046} C_VEL
LIN {X 0,Y 406.437,Z 568.01,A -85,B 0,C 180,E1 -10725.803,E2 -10725.803} C_VEL
LIN {X 0,Y 407.535,Z 558.731,A -85,B 0,C 180,E1 -10727.306,E2 -10727.306} C_VEL
LIN {X 0,Y 408.843,Z 547.383,A -85,B 0,C 180,E1 -10728.846,E2 -10728.846} C_VEL
LIN {X 0,Y 410.293,Z 534.464,A -85,B 0,C 180,E1 -10730.295,E2 -10730.295} C_VEL
LIN {X 0,Y 411.752,Z 520.928,A -85,B 0,C 180,E1 -10731.528,E2 -10731.528} C_VEL
LIN {X 0,Y 412.97,Z 507.615,A -85,B 0,C 180,E1 -10732.513,E2 -10732.513} C_VEL
LIN {X 0,Y 414.14,Z 492.366,A -85,B 0,C 180,E1 -10733.399,E2 -10733.399} C_VEL
LIN {X 0,Y 414.975,Z 477.478,A -85,B 0,C 180,E1 -10734.049,E2 -10734.049} C_VEL
LIN {X 0,Y 415.6,Z 462.192,A -85,B 0,C 180,E1 -10734.508,E2 -10734.508} C_VEL
LIN {X 0,Y 417.138,Z 383.214,A -85,B 0,C 180,E1 -10735.912,E2 -10735.912} C_VEL
LIN {X 0,Y 418.166,Z 326.035,A -85,B 0,C 180,E1 -10736.918,E2 -10736.918} C_VEL
LIN {X 0,Y 416.545,Z 320.085,A -85,B 0,C 180,E1 -10737.145,E2 -10737.145} C_VEL
LIN {X 0,Y 407.653,Z 299.871,A -85,B 0,C 180,E1 -10738.189,E2 -10738.189} C_VEL
LIN {X 0,Y 406.567,Z 297.314,A -85,B 0,C 180,E1 -10738.347,E2 -10738.347} C_VEL
LIN {X 0,Y 404.156,Z 287.771,A -85,B 0,C 180,E1 -10740.572,E2 -10740.572} C_VEL
LIN {X 0,Y 404.143,Z 287.772,A -85,B 0,C 180,E1 -10743.811,E2 -10743.811} C_VEL
LIN {X 0,Y 404.135,Z 287.77,A -85,B 0,C 180,E1 -10746.874,E2 -10746.874} C_VEL
LIN {X 0,Y 404.144,Z 287.762,A -85,B 0,C 180,E1 -10750.079,E2 -10750.079} C_VEL
LIN {X 0,Y 404.148,Z 287.769,A -85,B 0,C 180,E1 -10753.083,E2 -10753.083} C_VEL
LIN {X 0,Y 404.142,Z 287.768,A -85,B 0,C 180,E1 -10755.925,E2 -10755.925} C_VEL
LIN {X 0,Y 404.108,Z 287.759,A -85,B 0,C 180,E1 -10758.633,E2 -10758.633} C_VEL
LIN {X 0,Y 404.141,Z 287.765,A -85,B 0,C 180,E1 -10761.492,E2 -10761.492} C_VEL
LIN {X 0,Y 404.166,Z 287.76,A -85,B 0,C 180,E1 -10764.982,E2 -10764.982} C_VEL
LIN {X 0,Y 404.13,Z 287.758,A -85,B 0,C 180,E1 -10768.442,E2 -10768.442} C_VEL
LIN {X 0,Y 404.186,Z 287.76,A -85,B 0,C 180,E1 -10772,E2 -10772} C_VEL
LIN {X 0,Y 404.155,Z 287.767,A -85,B 0,C 180,E1 -10775.333,E2 -10775.333} C_VEL
LIN {X 0,Y 404.128,Z 287.765,A -85,B 0,C 180,E1 -10778.58,E2 -10778.58} C_VEL
LIN {X 0,Y 404.193,Z 287.755,A -85,B 0,C 180,E1 -10781.761,E2 -10781.761} C_VEL
LIN {X 0,Y 404.194,Z 287.764,A -85,B 0,C 180,E1 -10784.881,E2 -10784.881} C_VEL
LIN {X 0,Y 404.243,Z 287.752,A -85,B 0,C 180,E1 -10787.958,E2 -10787.958} C_VEL
LIN {X 0,Y 404.253,Z 287.749,A -85,B 0,C 180,E1 -10790.998,E2 -10790.998} C_VEL
LIN {X 0,Y 404.383,Z 287.736,A -85,B 0,C 180,E1 -10794.014,E2 -10794.014} C_VEL
LIN {X 0,Y 404.466,Z 287.726,A -85,B 0,C 180,E1 -10798.008,E2 -10798.008} C_VEL
LIN {X 0,Y 404.591,Z 287.706,A -85,B 0,C 180,E1 -10800,E2 -10800} C_VEL
LIN {X 0,Y 404.381,Z 287.737,A -85,B 0,C 180,E1 -10802.989,E2 -10802.989} C_VEL
LIN {X 0,Y 404.369,Z 287.74,A -85,B 0,C 180,E1 -10806.988,E2 -10806.988} C_VEL
LIN {X 0,Y 404.234,Z 287.757,A -85,B 0,C 180,E1 -10811.025,E2 -10811.025} C_VEL
LIN {X 0,Y 404.197,Z 287.756,A -85,B 0,C 180,E1 -10814.089,E2 -10814.089} C_VEL
LIN {X 0,Y 404.192,Z 287.757,A -85,B 0,C 180,E1 -10817.193,E2 -10817.193} C_VEL
LIN {X 0,Y 404.153,Z 287.771,A -85,B 0,C 180,E1 -10820.352,E2 -10820.352} C_VEL
LIN {X 0,Y 404.138,Z 287.768,A -85,B 0,C 180,E1 -10823.576,E2 -10823.576} C_VEL
LIN {X 0,Y 404.112,Z 287.771,A -85,B 0,C 180,E1 -10826.883,E2 -10826.883} C_VEL
LIN {X 0,Y 404.135,Z 287.771,A -85,B 0,C 180,E1 -10830.286,E2 -10830.286} C_VEL
LIN {X 0,Y 404.129,Z 287.765,A -85,B 0,C 180,E1 -10833.814,E2 -10833.814} C_VEL
LIN {X 0,Y 404.122,Z 287.768,A -85,B 0,C 180,E1 -10836.874,E2 -10836.874} C_VEL
LIN {X 0,Y 404.109,Z 287.758,A -85,B 0,C 180,E1 -10840.075,E2 -10840.075} C_VEL
LIN {X 0,Y 404.137,Z 287.768,A -85,B 0,C 180,E1 -10843.083,E2 -10843.083} C_VEL
LIN {X 0,Y 404.113,Z 287.773,A -85,B 0,C 180,E1 -10845.923,E2 -10845.923} C_VEL
LIN {X 0,Y 404.095,Z 287.773,A -85,B 0,C 180,E1 -10848.633,E2 -10848.633} C_VEL
LIN {X 0,Y 404.132,Z 287.768,A -85,B 0,C 180,E1 -10851.496,E2 -10851.496} C_VEL
LIN {X 0,Y 404.179,Z 287.765,A -85,B 0,C 180,E1 -10854.984,E2 -10854.984} C_VEL
LIN {X 0,Y 404.185,Z 287.805,A -85,B 0,C 180,E1 -10856.043,E2 -10856.043} C_VEL
LIN {X 0,Y 408.148,Z 303.137,A -85,B 0,C 180,E1 -10859.245,E2 -10859.245} C_VEL
LIN {X 0,Y 410.822,Z 315.386,A -85,B 0,C 180,E1 -10861.659,E2 -10861.659} C_VEL
LIN {X 0,Y 410.869,Z 317.65,A -85,B 0,C 180,E1 -10862.041,E2 -10862.041} C_VEL
LIN {X 0,Y 417.087,Z 348.646,A -85,B 0,C 180,E1 -10863.077,E2 -10863.077} C_VEL
LIN {X 0,Y 417.834,Z 354.261,A -85,B 0,C 180,E1 -10863.234,E2 -10863.234} C_VEL
LIN {X 0,Y 415.365,Z 481.801,A -85,B 0,C 180,E1 -10865.477,E2 -10865.477} C_VEL
LIN {X 0,Y 414.687,Z 496.989,A -85,B 0,C 180,E1 -10865.9,E2 -10865.9} C_VEL
LIN {X 0,Y 413.792,Z 510.383,A -85,B 0,C 180,E1 -10866.437,E2 -10866.437} C_VEL
LIN {X 0,Y 412.683,Z 524.789,A -85,B 0,C 180,E1 -10867.206,E2 -10867.206} C_VEL
LIN {X 0,Y 411.351,Z 539.098,A -85,B 0,C 180,E1 -10868.186,E2 -10868.186} C_VEL
LIN {X 0,Y 409.982,Z 552.129,A -85,B 0,C 180,E1 -10869.295,E2 -10869.295} C_VEL
LIN {X 0,Y 408.504,Z 565.24,A -85,B 0,C 180,E1 -10870.66,E2 -10870.66} C_VEL
LIN {X 0,Y 407.243,Z 577.113,A -85,B 0,C 180,E1 -10872.163,E2 -10872.163} C_VEL
LIN {X 0,Y 406.004,Z 587.103,A -85,B 0,C 180,E1 -10873.663,E2 -10873.663} C_VEL
LIN {X 0,Y 404.971,Z 596.883,A -85,B 0,C 180,E1 -10875.426,E2 -10875.426} C_VEL
LIN {X 0,Y 404.195,Z 605.049,A -85,B 0,C 180,E1 -10877.192,E2 -10877.192} C_VEL
LIN {X 0,Y 403.668,Z 611.802,A -85,B 0,C 180,E1 -10878.959,E2 -10878.959} C_VEL
LIN {X 0,Y 403.192,Z 618.039,A -85,B 0,C 180,E1 -10880.975,E2 -10880.975} C_VEL
LIN {X 0,Y 402.981,Z 622.868,A -85,B 0,C 180,E1 -10882.988,E2 -10882.988} C_VEL
LIN {X 0,Y 402.87,Z 626.406,A -85,B 0,C 180,E1 -10884.996,E2 -10884.996} C_VEL
LIN {X 0,Y 402.805,Z 628.732,A -85,B 0,C 180,E1 -10887,E2 -10887} C_VEL
LIN {X 0,Y 402.86,Z 629.905,A -85,B 0,C 180,E1 -10889,E2 -10889} C_VEL
LIN {X 0,Y 402.86,Z 629.904,A -85,B 0,C 180,E1 -10891,E2 -10891} C_VEL
LIN {X 0,Y 402.805,Z 628.724,A -85,B 0,C 180,E1 -10893,E2 -10893} C_VEL
LIN {X 0,Y 402.852,Z 626.393,A -85,B 0,C 180,E1 -10895.004,E2 -10895.004} C_VEL
LIN {X 0,Y 402.97,Z 622.857,A -85,B 0,C 180,E1 -10897.012,E2 -10897.012} C_VEL
LIN {X 0,Y 403.192,Z 618.028,A -85,B 0,C 180,E1 -10899.025,E2 -10899.025} C_VEL
LIN {X 0,Y 403.666,Z 611.778,A -85,B 0,C 180,E1 -10901.041,E2 -10901.041} C_VEL
LIN {X 0,Y 404.215,Z 603.927,A -85,B 0,C 180,E1 -10903.063,E2 -10903.063} C_VEL
LIN {X 0,Y 405.135,Z 595.589,A -85,B 0,C 180,E1 -10904.825,E2 -10904.825} C_VEL
LIN {X 0,Y 406.184,Z 585.542,A -85,B 0,C 180,E1 -10906.588,E2 -10906.588} C_VEL
LIN {X 0,Y 407.451,Z 575.276,A -85,B 0,C 180,E1 -10908.087,E2 -10908.087} C_VEL
LIN {X 0,Y 408.756,Z 563.041,A -85,B 0,C 180,E1 -10909.589,E2 -10909.589} C_VEL
LIN {X 0,Y 410.318,Z 549.43,A -85,B 0,C 180,E1 -10910.949,E2 -10910.949} C_VEL
LIN {X 0,Y 411.706,Z 535.785,A -85,B 0,C 180,E1 -10912.058,E2 -10912.058} C_VEL
LIN {X 0,Y 412.964,Z 521.654,A -85,B 0,C 180,E1 -10912.976,E2 -10912.976} C_VEL
LIN {X 0,Y 414.045,Z 507.22,A -85,B 0,C 180,E1 -10913.702,E2 -10913.702} C_VEL
LIN {X 0,Y 414.904,Z 492.2,A -85,B 0,C 180,E1 -10914.252,E2 -10914.252} C_VEL
LIN {X 0,Y 415.451,Z 476.917,A -85,B 0,C 180,E1 -10914.617,E2 -10914.617} C_VEL
LIN {X 0,Y 417.809,Z 353.897,A -85,B 0,C 180,E1 -10916.766,E2 -10916.766} C_VEL
LIN {X 0,Y 416.554,Z 346.135,A -85,B 0,C 180,E1 -10916.999,E2 -10916.999} C_VEL
LIN {X 0,Y 410.825,Z 317.358,A -85,B 0,C 180,E1 -10917.977,E2 -10917.977} C_VEL
LIN {X 0,Y 410.58,Z 313.761,A -85,B 0,C 180,E1 -10918.638,E2 -10918.638} C_VEL
LIN {X 0,Y 407.329,Z 299.926,A -85,B 0,C 180,E1 -10921.398,E2 -10921.398} C_VEL
LIN {X 0,Y 404.156,Z 287.765,A -85,B 0,C 180,E1 -10923.96,E2 -10923.96} C_VEL
LIN {X 0,Y 404.127,Z 287.771,A -85,B 0,C 180,E1 -10926.873,E2 -10926.873} C_VEL
LIN {X 0,Y 404.111,Z 287.775,A -85,B 0,C 180,E1 -10930.074,E2 -10930.074} C_VEL
LIN {X 0,Y 404.135,Z 287.769,A -85,B 0,C 180,E1 -10933.081,E2 -10933.081} C_VEL
LIN {X 0,Y 404.138,Z 287.772,A -85,B 0,C 180,E1 -10935.925,E2 -10935.925} C_VEL
LIN {X 0,Y 404.096,Z 287.773,A -85,B 0,C 180,E1 -10938.632,E2 -10938.632} C_VEL
LIN {X 0,Y 404.129,Z 287.771,A -85,B 0,C 180,E1 -10941.495,E2 -10941.495} C_VEL
LIN {X 0,Y 404.163,Z 287.761,A -85,B 0,C 180,E1 -10944.982,E2 -10944.982} C_VEL
LIN {X 0,Y 404.129,Z 287.768,A -85,B 0,C 180,E1 -10948.442,E2 -10948.442} C_VEL
LIN {X 0,Y 404.142,Z 287.765,A -85,B 0,C 180,E1 -10950.862,E2 -10950.862} C_VEL
LIN {X 0,Y 404.142,Z 287.766,A -85,B 0,C 180,E1 -10954.722,E2 -10954.722} C_VEL
LIN {X 0,Y 404.155,Z 287.768,A -85,B 0,C 180,E1 -10957.507,E2 -10957.507} C_VEL
LIN {X 0,Y 404.15,Z 287.749,A -85,B 0,C 180,E1 -10960.707,E2 -10960.707} C_VEL
LIN {X 0,Y 404.208,Z 287.762,A -85,B 0,C 180,E1 -10963.848,E2 -10963.848} C_VEL
LIN {X 0,Y 404.272,Z 287.744,A -85,B 0,C 180,E1 -10966.939,E2 -10966.939} C_VEL
LIN {X 0,Y 404.228,Z 287.747,A -85,B 0,C 180,E1 -10969.988,E2 -10969.988} C_VEL
LIN {X 0,Y 404.358,Z 287.741,A -85,B 0,C 180,E1 -10973.012,E2 -10973.012} C_VEL
LIN {X 0,Y 404.252,Z 287.748,A -85,B 0,C 180,E1 -10975.013,E2 -10975.013} C_VEL
LIN {X 0,Y 404.459,Z 287.722,A -85,B 0,C 180,E1 -10978.009,E2 -10978.009} C_VEL
LIN {X 0,Y 404.463,Z 287.722,A -85,B 0,C 180,E1 -10981.992,E2 -10981.992} C_VEL
LIN {X 0,Y 404.361,Z 287.735,A -85,B 0,C 180,E1 -10986.596,E2 -10986.596} C_VEL
LIN {X 0,Y 404.253,Z 287.755,A -85,B 0,C 180,E1 -10989.002,E2 -10989.002} C_VEL
LIN {X 0,Y 404.243,Z 287.753,A -85,B 0,C 180,E1 -10992.042,E2 -10992.042} C_VEL
LIN {X 0,Y 404.192,Z 287.759,A -85,B 0,C 180,E1 -10995.119,E2 -10995.119} C_VEL
LIN {X 0,Y 404.193,Z 287.757,A -85,B 0,C 180,E1 -10998.239,E2 -10998.239} C_VEL
LIN {X 0,Y 404.128,Z 287.755,A -85,B 0,C 180,E1 -11001.42,E2 -11001.42} C_VEL
LIN {X 0,Y 404.158,Z 287.767,A -85,B 0,C 180,E1 -11004.667,E2 -11004.667} C_VEL
LIN {X 0,Y 404.186,Z 287.748,A -85,B 0,C 180,E1 -11008,E2 -11008} C_VEL
LIN {X 0,Y 404.13,Z 287.765,A -85,B 0,C 180,E1 -11011.558,E2 -11011.558} C_VEL
LIN {X 0,Y 404.166,Z 287.764,A -85,B 0,C 180,E1 -11015.018,E2 -11015.018} C_VEL
LIN {X 0,Y 404.144,Z 287.769,A -85,B 0,C 180,E1 -11018.758,E2 -11018.758} C_VEL
LIN {X 0,Y 404.116,Z 287.769,A -85,B 0,C 180,E1 -11021.6,E2 -11021.6} C_VEL
LIN {X 0,Y 404.14,Z 287.769,A -85,B 0,C 180,E1 -11024.523,E2 -11024.523} C_VEL
LIN {X 0,Y 404.131,Z 287.771,A -85,B 0,C 180,E1 -11027.296,E2 -11027.296} C_VEL
LIN {X 0,Y 404.165,Z 287.766,A -85,B 0,C 180,E1 -11029.956,E2 -11029.956} C_VEL
LIN {X 0,Y 404.133,Z 287.769,A -85,B 0,C 180,E1 -11033.126,E2 -11033.126} C_VEL
LIN {X 0,Y 404.142,Z 287.767,A -85,B 0,C 180,E1 -11036.189,E2 -11036.189} C_VEL
LIN {X 0,Y 404.176,Z 287.828,A -85,B 0,C 180,E1 -11039.574,E2 -11039.574} C_VEL
LIN {X 0,Y 406.597,Z 297.377,A -85,B 0,C 180,E1 -11041.767,E2 -11041.767} C_VEL
LIN {X 0,Y 415.236,Z 316.975,A -85,B 0,C 180,E1 -11042.801,E2 -11042.801} C_VEL
LIN {X 0,Y 417.377,Z 322.656,A -85,B 0,C 180,E1 -11043.061,E2 -11043.061} C_VEL
LIN {X 0,Y 418.171,Z 326.363,A -85,B 0,C 180,E1 -11043.187,E2 -11043.187} C_VEL
LIN {X 0,Y 416.072,Z 438.698,A -85,B 0,C 180,E1 -11045.155,E2 -11045.155} C_VEL
LIN {X 0,Y 415.502,Z 463.438,A -85,B 0,C 180,E1 -11045.619,E2 -11045.619} C_VEL
LIN {X 0,Y 414.908,Z 478.304,A -85,B 0,C 180,E1 -11046.079,E2 -11046.079} C_VEL
LIN {X 0,Y 414.126,Z 493.083,A -85,B 0,C 180,E1 -11046.737,E2 -11046.737} C_VEL
LIN {X 0,Y 412.884,Z 508.063,A -85,B 0,C 180,E1 -11047.614,E2 -11047.614} C_VEL
LIN {X 0,Y 411.67,Z 521.314,A -85,B 0,C 180,E1 -11048.598,E2 -11048.598} C_VEL
LIN {X 0,Y 410.241,Z 534.778,A -85,B 0,C 180,E1 -11049.833,E2 -11049.833} C_VEL
LIN {X 0,Y 408.926,Z 547.101,A -85,B 0,C 180,E1 -11051.217,E2 -11051.217} C_VEL
LIN {X 0,Y 407.604,Z 558.107,A -85,B 0,C 180,E1 -11052.697,E2 -11052.697} C_VEL
LIN {X 0,Y 406.335,Z 568.904,A -85,B 0,C 180,E1 -11054.45,E2 -11054.45} C_VEL
LIN {X 0,Y 405.223,Z 578.011,A -85,B 0,C 180,E1 -11056.237,E2 -11056.237} C_VEL
LIN {X 0,Y 404.58,Z 585.282,A -85,B 0,C 180,E1 -11057.969,E2 -11057.969} C_VEL
LIN {X 0,Y 403.811,Z 592.221,A -85,B 0,C 180,E1 -11059.977,E2 -11059.977} C_VEL
LIN {X 0,Y 403.782,Z 592.508,A -85,B 0,C 180,E1 -11060.074,E2 -11060.074} C_VEL
LIN {X 0,Y 402.923,Z 594.8,A -85,B 0,C 180,E1 -11060.841,E2 -11060.841} C_VEL
LIN {X 0,Y 399.819,Z 598.206,A -85,B 0,C 180,E1 -11062.096,E2 -11062.096} C_VEL
LIN {X 0,Y 397.257,Z 600.552,A -85,B 0,C 180,E1 -11063.126,E2 -11063.126} C_VEL
LIN {X 0,Y 396.127,Z 602.069,A -85,B 0,C 180,E1 -11063.939,E2 -11063.939} C_VEL
LIN {X 0,Y 396.015,Z 602.498,A -85,B 0,C 180,E1 -11064.217,E2 -11064.217} C_VEL
LIN {X 0,Y 395.832,Z 604.878,A -85,B 0,C 180,E1 -11065.928,E2 -11065.928} C_VEL
LIN {X 0,Y 395.837,Z 606.615,A -85,B 0,C 180,E1 -11067.965,E2 -11067.965} C_VEL
LIN {X 0,Y 395.777,Z 607.224,A -85,B 0,C 180,E1 -11070,E2 -11070} C_VEL
LIN {X 0,Y 395.836,Z 606.662,A -85,B 0,C 180,E1 -11072.035,E2 -11072.035} C_VEL
LIN {X 0,Y 395.824,Z 604.989,A -85,B 0,C 180,E1 -11074.073,E2 -11074.073} C_VEL
LIN {X 0,Y 396.028,Z 602.156,A -85,B 0,C 180,E1 -11076.112,E2 -11076.112} C_VEL
LIN {X 0,Y 396.314,Z 598.103,A -85,B 0,C 180,E1 -11078.156,E2 -11078.156} C_VEL
LIN {X 0,Y 396.771,Z 592.726,A -85,B 0,C 180,E1 -11080.202,E2 -11080.202} C_VEL
LIN {X 0,Y 397.584,Z 585.869,A -85,B 0,C 180,E1 -11082.246,E2 -11082.246} C_VEL
LIN {X 0,Y 398.222,Z 579.06,A -85,B 0,C 180,E1 -11083.912,E2 -11083.912} C_VEL
LIN {X 0,Y 399.207,Z 570.958,A -85,B 0,C 180,E1 -11085.573,E2 -11085.573} C_VEL
LIN {X 0,Y 400.514,Z 560.55,A -85,B 0,C 180,E1 -11087.355,E2 -11087.355} C_VEL
LIN {X 0,Y 401.907,Z 549.389,A -85,B 0,C 180,E1 -11088.938,E2 -11088.938} C_VEL
LIN {X 0,Y 403.336,Z 537.009,A -85,B 0,C 180,E1 -11090.395,E2 -11090.395} C_VEL
LIN {X 0,Y 404.833,Z 523.999,A -85,B 0,C 180,E1 -11091.647,E2 -11091.647} C_VEL
LIN {X 0,Y 406.086,Z 511.335,A -85,B 0,C 180,E1 -11092.648,E2 -11092.648} C_VEL
LIN {X 0,Y 407.279,Z 497.818,A -85,B 0,C 180,E1 -11093.506,E2 -11093.506} C_VEL
LIN {X 0,Y 408.194,Z 482.782,A -85,B 0,C 180,E1 -11094.249,E2 -11094.249} C_VEL
LIN {X 0,Y 408.912,Z 468.12,A -85,B 0,C 180,E1 -11094.767,E2 -11094.767} C_VEL
LIN {X 0,Y 409.492,Z 451.294,A -85,B 0,C 180,E1 -11095.136,E2 -11095.136} C_VEL
LIN {X 0,Y 411.9,Z 328.236,A -85,B 0,C 180,E1 -11097.323,E2 -11097.323} C_VEL
LIN {X 0,Y 410.811,Z 323.397,A -85,B 0,C 180,E1 -11097.495,E2 -11097.495} C_VEL
LIN {X 0,Y 401.703,Z 302.708,A -85,B 0,C 180,E1 -11098.591,E2 -11098.591} C_VEL
LIN {X 0,Y 399.405,Z 297.598,A -85,B 0,C 180,E1 -11098.89,E2 -11098.89} C_VEL
LIN {X 0,Y 397.121,Z 288.647,A -85,B 0,C 180,E1 -11101.026,E2 -11101.026} C_VEL
LIN {X 0,Y 397.123,Z 288.643,A -85,B 0,C 180,E1 -11104.492,E2 -11104.492} C_VEL
LIN {X 0,Y 397.1,Z 288.649,A -85,B 0,C 180,E1 -11108.274,E2 -11108.274} C_VEL
LIN {X 0,Y 397.084,Z 288.641,A -85,B 0,C 180,E1 -11110.908,E2 -11110.908} C_VEL
LIN {X 0,Y 397.096,Z 288.648,A -85,B 0,C 180,E1 -11113.648,E2 -11113.648} C_VEL
LIN {X 0,Y 397.095,Z 288.645,A -85,B 0,C 180,E1 -11116.52,E2 -11116.52} C_VEL
LIN {X 0,Y 397.097,Z 288.644,A -85,B 0,C 180,E1 -11120.421,E2 -11120.421} C_VEL
LIN {X 0,Y 397.09,Z 288.633,A -85,B 0,C 180,E1 -11123.004,E2 -11123.004} C_VEL
LIN {X 0,Y 397.104,Z 288.646,A -85,B 0,C 180,E1 -11126.726,E2 -11126.726} C_VEL
LIN {X 0,Y 397.112,Z 288.629,A -85,B 0,C 180,E1 -11130.295,E2 -11130.295} C_VEL
LIN {X 0,Y 397.185,Z 288.634,A -85,B 0,C 180,E1 -11132.609,E2 -11132.609} C_VEL
LIN {X 0,Y 397.114,Z 288.641,A -85,B 0,C 180,E1 -11135.98,E2 -11135.98} C_VEL
LIN {X 0,Y 397.129,Z 288.64,A -85,B 0,C 180,E1 -11139.704,E2 -11139.704} C_VEL
LIN {X 0,Y 397.172,Z 288.632,A -85,B 0,C 180,E1 -11142.845,E2 -11142.845} C_VEL
LIN {X 0,Y 397.219,Z 288.626,A -85,B 0,C 180,E1 -11146.702,E2 -11146.702} C_VEL
LIN {X 0,Y 397.203,Z 288.629,A -85,B 0,C 180,E1 -11149.808,E2 -11149.808} C_VEL
LIN {X 0,Y 397.32,Z 288.621,A -85,B 0,C 180,E1 -11152.887,E2 -11152.887} C_VEL
LIN {X 0,Y 397.23,Z 288.623,A -85,B 0,C 180,E1 -11154.925,E2 -11154.925} C_VEL
LIN {X 0,Y 397.434,Z 288.602,A -85,B 0,C 180,E1 -11157.973,E2 -11157.973} C_VEL
LIN {X 0,Y 397.561,Z 288.581,A -85,B 0,C 180,E1 -11160,E2 -11160} C_VEL
LIN {X 0,Y 397.315,Z 288.617,A -85,B 0,C 180,E1 -11163.042,E2 -11163.042} C_VEL
LIN {X 0,Y 397.335,Z 288.613,A -85,B 0,C 180,E1 -11166.092,E2 -11166.092} C_VEL
LIN {X 0,Y 397.22,Z 288.624,A -85,B 0,C 180,E1 -11169.162,E2 -11169.162} C_VEL
LIN {X 0,Y 397.206,Z 288.635,A -85,B 0,C 180,E1 -11172.258,E2 -11172.258} C_VEL
LIN {X 0,Y 397.165,Z 288.637,A -85,B 0,C 180,E1 -11175.392,E2 -11175.392} C_VEL
LIN {X 0,Y 397.146,Z 288.639,A -85,B 0,C 180,E1 -11178.574,E2 -11178.574} C_VEL
LIN {X 0,Y 397.084,Z 288.645,A -85,B 0,C 180,E1 -11181.819,E2 -11181.819} C_VEL
LIN {X 0,Y 397.092,Z 288.643,A -85,B 0,C 180,E1 -11185.136,E2 -11185.136} C_VEL
LIN {X 0,Y 397.067,Z 288.651,A -85,B 0,C 180,E1 -11188.548,E2 -11188.548} C_VEL
LIN {X 0,Y 397.072,Z 288.65,A -85,B 0,C 180,E1 -11191.837,E2 -11191.837} C_VEL
LIN {X 0,Y 397.107,Z 288.646,A -85,B 0,C 180,E1 -11194.495,E2 -11194.495} C_VEL
LIN {X 0,Y 397.081,Z 288.647,A -85,B 0,C 180,E1 -11198.277,E2 -11198.277} C_VEL
LIN {X 0,Y 397.046,Z 288.644,A -85,B 0,C 180,E1 -11201.977,E2 -11201.977} C_VEL
LIN {X 0,Y 397.077,Z 288.647,A -85,B 0,C 180,E1 -11205.07,E2 -11205.07} C_VEL
LIN {X 0,Y 397.045,Z 288.651,A -85,B 0,C 180,E1 -11208.024,E2 -11208.024} C_VEL
LIN {X 0,Y 397.084,Z 288.646,A -85,B 0,C 180,E1 -11211.724,E2 -11211.724} C_VEL
LIN {X 0,Y 397.155,Z 288.739,A -85,B 0,C 180,E1 -11215.582,E2 -11215.582} C_VEL
LIN {X 0,Y 400.678,Z 302.343,A -85,B 0,C 180,E1 -11218.501,E2 -11218.501} C_VEL
LIN {X 0,Y 403.815,Z 315.825,A -85,B 0,C 180,E1 -11221.242,E2 -11221.242} C_VEL
LIN {X 0,Y 404.091,Z 317.395,A -85,B 0,C 180,E1 -11221.528,E2 -11221.528} C_VEL
LIN {X 0,Y 408.31,Z 336.941,A -85,B 0,C 180,E1 -11222.227,E2 -11222.227} C_VEL
LIN {X 0,Y 411.48,Z 354.654,A -85,B 0,C 180,E1 -11222.798,E2 -11222.798} C_VEL
LIN {X 0,Y 408.909,Z 481.614,A -85,B 0,C 180,E1 -11225.064,E2 -11225.064} C_VEL
LIN {X 0,Y 408.227,Z 496.797,A -85,B 0,C 180,E1 -11225.494,E2 -11225.494} C_VEL
LIN {X 0,Y 407.209,Z 511.281,A -85,B 0,C 180,E1 -11226.089,E2 -11226.089} C_VEL
LIN {X 0,Y 406.13,Z 524.591,A -85,B 0,C 180,E1 -11226.817,E2 -11226.817} C_VEL
LIN {X 0,Y 404.734,Z 538.898,A -85,B 0,C 180,E1 -11227.811,E2 -11227.811} C_VEL
LIN {X 0,Y 403.318,Z 551.929,A -85,B 0,C 180,E1 -11228.937,E2 -11228.937} C_VEL
LIN {X 0,Y 401.897,Z 563.964,A -85,B 0,C 180,E1 -11230.196,E2 -11230.196} C_VEL
LIN {X 0,Y 400.626,Z 575.118,A -85,B 0,C 180,E1 -11231.593,E2 -11231.593} C_VEL
LIN {X 0,Y 399.328,Z 585.38,A -85,B 0,C 180,E1 -11233.119,E2 -11233.119} C_VEL
LIN {X 0,Y 398.183,Z 595.418,A -85,B 0,C 180,E1 -11234.91,E2 -11234.91} C_VEL
LIN {X 0,Y 397.151,Z 604.569,A -85,B 0,C 180,E1 -11236.892,E2 -11236.892} C_VEL
LIN {X 0,Y 396.629,Z 611.598,A -85,B 0,C 180,E1 -11238.761,E2 -11238.761} C_VEL
LIN {X 0,Y 396.11,Z 617.835,A -85,B 0,C 180,E1 -11240.812,E2 -11240.812} C_VEL
LIN {X 0,Y 395.905,Z 622.664,A -85,B 0,C 180,E1 -11242.862,E2 -11242.862} C_VEL
LIN {X 0,Y 395.768,Z 626.202,A -85,B 0,C 180,E1 -11244.906,E2 -11244.906} C_VEL
LIN {X 0,Y 395.708,Z 628.53,A -85,B 0,C 180,E1 -11246.946,E2 -11246.946} C_VEL
LIN {X 0,Y 395.788,Z 629.703,A -85,B 0,C 180,E1 -11248.983,E2 -11248.983} C_VEL
LIN {X 0,Y 395.788,Z 629.701,A -85,B 0,C 180,E1 -11251.017,E2 -11251.017} C_VEL
LIN {X 0,Y 395.707,Z 628.521,A -85,B 0,C 180,E1 -11253.054,E2 -11253.054} C_VEL
LIN {X 0,Y 395.753,Z 626.189,A -85,B 0,C 180,E1 -11255.094,E2 -11255.094} C_VEL
LIN {X 0,Y 395.894,Z 622.653,A -85,B 0,C 180,E1 -11257.138,E2 -11257.138} C_VEL
LIN {X 0,Y 396.11,Z 617.822,A -85,B 0,C 180,E1 -11259.188,E2 -11259.188} C_VEL
LIN {X 0,Y 396.626,Z 611.571,A -85,B 0,C 180,E1 -11261.239,E2 -11261.239} C_VEL
LIN {X 0,Y 397.226,Z 603.618,A -85,B 0,C 180,E1 -11263.321,E2 -11263.321} C_VEL
LIN {X 0,Y 398.191,Z 595.381,A -85,B 0,C 180,E1 -11265.089,E2 -11265.089} C_VEL
LIN {X 0,Y 399.337,Z 585.336,A -85,B 0,C 180,E1 -11266.881,E2 -11266.881} C_VEL
LIN {X 0,Y 400.642,Z 575.068,A -85,B 0,C 180,E1 -11268.406,E2 -11268.406} C_VEL
LIN {X 0,Y 402.023,Z 562.833,A -85,B 0,C 180,E1 -11269.931,E2 -11269.931} C_VEL
LIN {X 0,Y 403.64,Z 549.222,A -85,B 0,C 180,E1 -11271.313,E2 -11271.313} C_VEL
LIN {X 0,Y 405.105,Z 535.576,A -85,B 0,C 180,E1 -11272.436,E2 -11272.436} C_VEL
LIN {X 0,Y 406.411,Z 521.444,A -85,B 0,C 180,E1 -11273.368,E2 -11273.368} C_VEL
LIN {X 0,Y 407.567,Z 506.223,A -85,B 0,C 180,E1 -11274.139,E2 -11274.139} C_VEL
LIN {X 0,Y 408.522,Z 490.968,A -85,B 0,C 180,E1 -11274.69,E2 -11274.69} C_VEL
LIN {X 0,Y 409.061,Z 475.006,A -85,B 0,C 180,E1 -11275.062,E2 -11275.062} C_VEL
LIN {X 0,Y 411.442,Z 354.841,A -85,B 0,C 180,E1 -11277.192,E2 -11277.192} C_VEL
LIN {X 0,Y 408.077,Z 335.896,A -85,B 0,C 180,E1 -11277.8,E2 -11277.8} C_VEL
LIN {X 0,Y 404.061,Z 317.281,A -85,B 0,C 180,E1 -11278.465,E2 -11278.465} C_VEL
LIN {X 0,Y 401.406,Z 305.061,A -85,B 0,C 180,E1 -11280.917,E2 -11280.917} C_VEL
LIN {X 0,Y 397.561,Z 290.397,A -85,B 0,C 180,E1 -11284.043,E2 -11284.043} C_VEL
LIN {X 0,Y 397.126,Z 288.644,A -85,B 0,C 180,E1 -11284.441,E2 -11284.441} C_VEL
LIN {X 0,Y 397.084,Z 288.649,A -85,B 0,C 180,E1 -11288.276,E2 -11288.276} C_VEL
LIN {X 0,Y 397.045,Z 288.656,A -85,B 0,C 180,E1 -11291.976,E2 -11291.976} C_VEL
LIN {X 0,Y 397.077,Z 288.647,A -85,B 0,C 180,E1 -11295.069,E2 -11295.069} C_VEL
LIN {X 0,Y 397.046,Z 288.655,A -85,B 0,C 180,E1 -11298.023,E2 -11298.023} C_VEL
LIN {X 0,Y 397.081,Z 288.647,A -85,B 0,C 180,E1 -11301.723,E2 -11301.723} C_VEL
LIN {X 0,Y 397.107,Z 288.643,A -85,B 0,C 180,E1 -11305.505,E2 -11305.505} C_VEL
LIN {X 0,Y 397.068,Z 288.647,A -85,B 0,C 180,E1 -11309.117,E2 -11309.117} C_VEL
LIN {X 0,Y 397.071,Z 288.645,A -85,B 0,C 180,E1 -11312.246,E2 -11312.246} C_VEL
LIN {X 0,Y 397.092,Z 288.644,A -85,B 0,C 180,E1 -11314.864,E2 -11314.864} C_VEL
LIN {X 0,Y 397.084,Z 288.645,A -85,B 0,C 180,E1 -11318.181,E2 -11318.181} C_VEL
LIN {X 0,Y 397.145,Z 288.62,A -85,B 0,C 180,E1 -11321.426,E2 -11321.426} C_VEL
LIN {X 0,Y 397.165,Z 288.635,A -85,B 0,C 180,E1 -11324.608,E2 -11324.608} C_VEL
LIN {X 0,Y 397.201,Z 288.609,A -85,B 0,C 180,E1 -11327.741,E2 -11327.741} C_VEL
LIN {X 0,Y 397.213,Z 288.624,A -85,B 0,C 180,E1 -11330.837,E2 -11330.837} C_VEL
LIN {X 0,Y 397.332,Z 288.61,A -85,B 0,C 180,E1 -11333.908,E2 -11333.908} C_VEL
LIN {X 0,Y 397.428,Z 288.598,A -85,B 0,C 180,E1 -11337.973,E2 -11337.973} C_VEL
LIN {X 0,Y 397.432,Z 288.598,A -85,B 0,C 180,E1 -11342.027,E2 -11342.027} C_VEL
LIN {X 0,Y 397.312,Z 288.612,A -85,B 0,C 180,E1 -11346.593,E2 -11346.593} C_VEL
LIN {X 0,Y 397.223,Z 288.633,A -85,B 0,C 180,E1 -11349.163,E2 -11349.163} C_VEL
LIN {X 0,Y 397.207,Z 288.629,A -85,B 0,C 180,E1 -11352.259,E2 -11352.259} C_VEL
LIN {X 0,Y 397.166,Z 288.635,A -85,B 0,C 180,E1 -11355.393,E2 -11355.393} C_VEL
LIN {X 0,Y 397.147,Z 288.636,A -85,B 0,C 180,E1 -11358.574,E2 -11358.574} C_VEL
LIN {X 0,Y 397.086,Z 288.637,A -85,B 0,C 180,E1 -11361.819,E2 -11361.819} C_VEL
LIN {X 0,Y 397.118,Z 288.641,A -85,B 0,C 180,E1 -11365.134,E2 -11365.134} C_VEL
LIN {X 0,Y 397.153,Z 288.622,A -85,B 0,C 180,E1 -11367.776,E2 -11367.776} C_VEL
LIN {X 0,Y 397.07,Z 288.652,A -85,B 0,C 180,E1 -11370.883,E2 -11370.883} C_VEL
LIN {X 0,Y 397.11,Z 288.644,A -85,B 0,C 180,E1 -11374.495,E2 -11374.495} C_VEL
LIN {X 0,Y 397.093,Z 288.642,A -85,B 0,C 180,E1 -11378.276,E2 -11378.276} C_VEL
LIN {X 0,Y 397.082,Z 288.648,A -85,B 0,C 180,E1 -11380.91,E2 -11380.91} C_VEL
LIN {X 0,Y 397.095,Z 288.644,A -85,B 0,C 180,E1 -11383.649,E2 -11383.649} C_VEL
LIN {X 0,Y 397.097,Z 288.647,A -85,B 0,C 180,E1 -11386.522,E2 -11386.522} C_VEL
LIN {X 0,Y 397.111,Z 288.642,A -85,B 0,C 180,E1 -11390.424,E2 -11390.424} C_VEL
LIN {X 0,Y 397.104,Z 288.639,A -85,B 0,C 180,E1 -11394.266,E2 -11394.266} C_VEL
LIN {X 0,Y 397.112,Z 288.64,A -85,B 0,C 180,E1 -11396.728,E2 -11396.728} C_VEL
LIN {X 0,Y 397.119,Z 288.721,A -85,B 0,C 180,E1 -11399.122,E2 -11399.122} C_VEL
LIN {X 0,Y 399.471,Z 297.881,A -85,B 0,C 180,E1 -11401.238,E2 -11401.238} C_VEL
LIN {X 0,Y 408.015,Z 316.715,A -85,B 0,C 180,E1 -11402.269,E2 -11402.269} C_VEL
LIN {X 0,Y 411.345,Z 325.189,A -85,B 0,C 180,E1 -11402.678,E2 -11402.678} C_VEL
LIN {X 0,Y 411.873,Z 329.005,A -85,B 0,C 180,E1 -11402.79,E2 -11402.79} C_VEL
LIN {X 0,Y 409.658,Z 438.926,A -85,B 0,C 180,E1 -11404.739,E2 -11404.739} C_VEL
LIN {X 0,Y 409.05,Z 463.657,A -85,B 0,C 180,E1 -11405.208,E2 -11405.208} C_VEL
LIN {X 0,Y 408.441,Z 478.64,A -85,B 0,C 180,E1 -11405.681,E2 -11405.681} C_VEL
LIN {X 0,Y 407.639,Z 492.606,A -85,B 0,C 180,E1 -11406.306,E2 -11406.306} C_VEL
LIN {X 0,Y 406.513,Z 506.387,A -85,B 0,C 180,E1 -11407.109,E2 -11407.109} C_VEL
LIN {X 0,Y 405.19,Z 519.964,A -85,B 0,C 180,E1 -11408.105,E2 -11408.105} C_VEL
LIN {X 0,Y 403.712,Z 533.735,A -85,B 0,C 180,E1 -11409.359,E2 -11409.359} C_VEL
LIN {X 0,Y 402.383,Z 545.09,A -85,B 0,C 180,E1 -11410.619,E2 -11410.619} C_VEL
LIN {X 0,Y 401.013,Z 556.547,A -85,B 0,C 180,E1 -11412.14,E2 -11412.14} C_VEL
LIN {X 0,Y 399.796,Z 566.186,A -85,B 0,C 180,E1 -11413.665,E2 -11413.665} C_VEL
LIN {X 0,Y 398.646,Z 575.631,A -85,B 0,C 180,E1 -11415.451,E2 -11415.451} C_VEL
LIN {X 0,Y 397.789,Z 583.49,A -85,B 0,C 180,E1 -11417.242,E2 -11417.242} C_VEL
LIN {X 0,Y 396.935,Z 590.827,A -85,B 0,C 180,E1 -11419.286,E2 -11419.286} C_VEL
LIN {X 0,Y 396.448,Z 596.645,A -85,B 0,C 180,E1 -11421.334,E2 -11421.334} C_VEL
LIN {X 0,Y 396.13,Z 601.28,A -85,B 0,C 180,E1 -11423.481,E2 -11423.481} C_VEL
LIN {X 0,Y 396.015,Z 602.498,A -85,B 0,C 180,E1 -11424.217,E2 -11424.217} C_VEL
LIN {X 0,Y 395.271,Z 603.816,A -85,B 0,C 180,E1 -11425.045,E2 -11425.045} C_VEL
LIN {X 0,Y 392.307,Z 605.528,A -85,B 0,C 180,E1 -11426.4,E2 -11426.4} C_VEL
LIN {X 0,Y 389.842,Z 606.519,A -85,B 0,C 180,E1 -11427.501,E2 -11427.501} C_VEL
LIN {X 0,Y 388.796,Z 607.013,A -85,B 0,C 180,E1 -11428.359,E2 -11428.359} C_VEL
LIN {X 0,Y 388.716,Z 607.131,A -85,B 0,C 180,E1 -11428.649,E2 -11428.649} C_VEL
LIN {X 0,Y 388.706,Z 607.426,A -85,B 0,C 180,E1 -11430,E2 -11430} C_VEL
LIN {X 0,Y 388.738,Z 606.865,A -85,B 0,C 180,E1 -11432.072,E2 -11432.072} C_VEL
LIN {X 0,Y 388.751,Z 605.191,A -85,B 0,C 180,E1 -11434.147,E2 -11434.147} C_VEL
LIN {X 0,Y 388.962,Z 602.359,A -85,B 0,C 180,E1 -11436.224,E2 -11436.224} C_VEL
LIN {X 0,Y 389.262,Z 598.305,A -85,B 0,C 180,E1 -11438.304,E2 -11438.304} C_VEL
LIN {X 0,Y 389.759,Z 592.928,A -85,B 0,C 180,E1 -11440.388,E2 -11440.388} C_VEL
LIN {X 0,Y 390.604,Z 586.071,A -85,B 0,C 180,E1 -11442.469,E2 -11442.469} C_VEL
LIN {X 0,Y 391.308,Z 579.193,A -85,B 0,C 180,E1 -11444.179,E2 -11444.179} C_VEL
LIN {X 0,Y 392.353,Z 571.159,A -85,B 0,C 180,E1 -11445.852,E2 -11445.852} C_VEL
LIN {X 0,Y 393.702,Z 560.751,A -85,B 0,C 180,E1 -11447.665,E2 -11447.665} C_VEL
LIN {X 0,Y 395.125,Z 549.962,A -85,B 0,C 180,E1 -11449.224,E2 -11449.224} C_VEL
LIN {X 0,Y 396.529,Z 538.376,A -85,B 0,C 180,E1 -11450.625,E2 -11450.625} C_VEL
LIN {X 0,Y 398.086,Z 525.616,A -85,B 0,C 180,E1 -11451.897,E2 -11451.897} C_VEL
LIN {X 0,Y 399.391,Z 513.292,A -85,B 0,C 180,E1 -11452.912,E2 -11452.912} C_VEL
LIN {X 0,Y 400.578,Z 500.065,A -85,B 0,C 180,E1 -11453.798,E2 -11453.798} C_VEL
LIN {X 0,Y 401.615,Z 484.853,A -85,B 0,C 180,E1 -11454.587,E2 -11454.587} C_VEL
LIN {X 0,Y 402.45,Z 469.444,A -85,B 0,C 180,E1 -11455.157,E2 -11455.157} C_VEL
LIN {X 0,Y 403.056,Z 453.258,A -85,B 0,C 180,E1 -11455.531,E2 -11455.531} C_VEL
LIN {X 0,Y 405.602,Z 328.768,A -85,B 0,C 180,E1 -11457.776,E2 -11457.776} C_VEL
LIN {X 0,Y 404.076,Z 324.3,A -85,B 0,C 180,E1 -11457.979,E2 -11457.979} C_VEL
LIN {X 0,Y 395.394,Z 304.66,A -85,B 0,C 180,E1 -11459.054,E2 -11459.054} C_VEL
LIN {X 0,Y 392.167,Z 297.772,A -85,B 0,C 180,E1 -11459.486,E2 -11459.486} C_VEL
LIN {X 0,Y 390.066,Z 289.527,A -85,B 0,C 180,E1 -11461.5,E2 -11461.5} C_VEL
LIN {X 0,Y 390.083,Z 289.523,A -85,B 0,C 180,E1 -11465.206,E2 -11465.206} C_VEL
LIN {X 0,Y 390.086,Z 289.524,A -85,B 0,C 180,E1 -11469.092,E2 -11469.092} C_VEL
LIN {X 0,Y 390.038,Z 289.526,A -85,B 0,C 180,E1 -11472.373,E2 -11472.373} C_VEL
LIN {X 0,Y 390.039,Z 289.526,A -85,B 0,C 180,E1 -11475.353,E2 -11475.353} C_VEL
LIN {X 0,Y 390.021,Z 289.512,A -85,B 0,C 180,E1 -11478.185,E2 -11478.185} C_VEL
LIN {X 0,Y 390.076,Z 289.522,A -85,B 0,C 180,E1 -11480.906,E2 -11480.906} C_VEL
LIN {X 0,Y 390.062,Z 289.514,A -85,B 0,C 180,E1 -11484.791,E2 -11484.791} C_VEL
LIN {X 0,Y 390.014,Z 289.514,A -85,B 0,C 180,E1 -11488.495,E2 -11488.495} C_VEL
LIN {X 0,Y 390.11,Z 289.513,A -85,B 0,C 180,E1 -11492.069,E2 -11492.069} C_VEL
LIN {X 0,Y 390.053,Z 289.523,A -85,B 0,C 180,E1 -11495.517,E2 -11495.517} C_VEL
LIN {X 0,Y 390.046,Z 289.52,A -85,B 0,C 180,E1 -11498.877,E2 -11498.877} C_VEL
LIN {X 0,Y 390.101,Z 289.511,A -85,B 0,C 180,E1 -11502.165,E2 -11502.165} C_VEL
LIN {X 0,Y 390.132,Z 289.509,A -85,B 0,C 180,E1 -11505.392,E2 -11505.392} C_VEL
LIN {X 0,Y 390.134,Z 289.513,A -85,B 0,C 180,E1 -11508.571,E2 -11508.571} C_VEL
LIN {X 0,Y 390.259,Z 289.492,A -85,B 0,C 180,E1 -11512.072,E2 -11512.072} C_VEL
LIN {X 0,Y 390.202,Z 289.499,A -85,B 0,C 180,E1 -11514.833,E2 -11514.833} C_VEL
LIN {X 0,Y 390.402,Z 289.478,A -85,B 0,C 180,E1 -11517.937,E2 -11517.937} C_VEL
LIN {X 0,Y 390.531,Z 289.457,A -85,B 0,C 180,E1 -11520,E2 -11520} C_VEL
LIN {X 0,Y 390.251,Z 289.496,A -85,B 0,C 180,E1 -11523.097,E2 -11523.097} C_VEL
LIN {X 0,Y 390.29,Z 289.492,A -85,B 0,C 180,E1 -11526.202,E2 -11526.202} C_VEL
LIN {X 0,Y 390.178,Z 289.501,A -85,B 0,C 180,E1 -11529.329,E2 -11529.329} C_VEL
LIN {X 0,Y 390.158,Z 289.509,A -85,B 0,C 180,E1 -11532.483,E2 -11532.483} C_VEL
LIN {X 0,Y 390.126,Z 289.514,A -85,B 0,C 180,E1 -11535.677,E2 -11535.677} C_VEL
LIN {X 0,Y 390.091,Z 289.519,A -85,B 0,C 180,E1 -11538.923,E2 -11538.923} C_VEL
LIN {X 0,Y 390.024,Z 289.524,A -85,B 0,C 180,E1 -11542.235,E2 -11542.235} C_VEL
LIN {X 0,Y 390.04,Z 289.521,A -85,B 0,C 180,E1 -11545.723,E2 -11545.723} C_VEL
LIN {X 0,Y 390.022,Z 289.525,A -85,B 0,C 180,E1 -11549.112,E2 -11549.112} C_VEL
LIN {X 0,Y 390.032,Z 289.519,A -85,B 0,C 180,E1 -11552.722,E2 -11552.722} C_VEL
LIN {X 0,Y 390.032,Z 289.525,A -85,B 0,C 180,E1 -11555.823,E2 -11555.823} C_VEL
LIN {X 0,Y 390.028,Z 289.521,A -85,B 0,C 180,E1 -11559.213,E2 -11559.213} C_VEL
LIN {X 0,Y 390.025,Z 289.525,A -85,B 0,C 180,E1 -11562.373,E2 -11562.373} C_VEL
LIN {X 0,Y 390.033,Z 289.526,A -85,B 0,C 180,E1 -11565.354,E2 -11565.354} C_VEL
LIN {X 0,Y 390.008,Z 289.527,A -85,B 0,C 180,E1 -11568.185,E2 -11568.185} C_VEL
LIN {X 0,Y 390.051,Z 289.522,A -85,B 0,C 180,E1 -11570.904,E2 -11570.904} C_VEL
LIN {X 0,Y 390.084,Z 289.521,A -85,B 0,C 180,E1 -11574.794,E2 -11574.794} C_VEL
LIN {X 0,Y 390.083,Z 289.625,A -85,B 0,C 180,E1 -11575.087,E2 -11575.087} C_VEL
LIN {X 0,Y 393.469,Z 302.365,A -85,B 0,C 180,E1 -11577.902,E2 -11577.902} C_VEL
LIN {X 0,Y 396.701,Z 316.284,A -85,B 0,C 180,E1 -11580.805,E2 -11580.805} C_VEL
LIN {X 0,Y 397.01,Z 317.385,A -85,B 0,C 180,E1 -11580.976,E2 -11580.976} C_VEL
LIN {X 0,Y 398.858,Z 322.74,A -85,B 0,C 180,E1 -11581.23,E2 -11581.23} C_VEL
LIN {X 0,Y 404.858,Z 353.195,A -85,B 0,C 180,E1 -11582.29,E2 -11582.29} C_VEL
LIN {X 0,Y 405.109,Z 357.317,A -85,B 0,C 180,E1 -11582.39,E2 -11582.39} C_VEL
LIN {X 0,Y 402.492,Z 481.428,A -85,B 0,C 180,E1 -11584.638,E2 -11584.638} C_VEL
LIN {X 0,Y 401.77,Z 496.603,A -85,B 0,C 180,E1 -11585.074,E2 -11585.074} C_VEL
LIN {X 0,Y 400.732,Z 510.515,A -85,B 0,C 180,E1 -11585.648,E2 -11585.648} C_VEL
LIN {X 0,Y 399.6,Z 524.393,A -85,B 0,C 180,E1 -11586.415,E2 -11586.415} C_VEL
LIN {X 0,Y 398.135,Z 538.699,A -85,B 0,C 180,E1 -11587.423,E2 -11587.423} C_VEL
LIN {X 0,Y 396.667,Z 551.728,A -85,B 0,C 180,E1 -11588.567,E2 -11588.567} C_VEL
LIN {X 0,Y 395.158,Z 563.762,A -85,B 0,C 180,E1 -11589.844,E2 -11589.844} C_VEL
LIN {X 0,Y 393.802,Z 574.914,A -85,B 0,C 180,E1 -11591.263,E2 -11591.263} C_VEL
LIN {X 0,Y 392.463,Z 585.177,A -85,B 0,C 180,E1 -11592.815,E2 -11592.815} C_VEL
LIN {X 0,Y 391.263,Z 595.215,A -85,B 0,C 180,E1 -11594.637,E2 -11594.637} C_VEL
LIN {X 0,Y 390.215,Z 603.932,A -85,B 0,C 180,E1 -11596.549,E2 -11596.549} C_VEL
LIN {X 0,Y 389.6,Z 611.394,A -85,B 0,C 180,E1 -11598.555,E2 -11598.555} C_VEL
LIN {X 0,Y 389.04,Z 617.631,A -85,B 0,C 180,E1 -11600.643,E2 -11600.643} C_VEL
LIN {X 0,Y 388.825,Z 622.461,A -85,B 0,C 180,E1 -11602.731,E2 -11602.731} C_VEL
LIN {X 0,Y 388.673,Z 625.999,A -85,B 0,C 180,E1 -11604.813,E2 -11604.813} C_VEL
LIN {X 0,Y 388.615,Z 628.327,A -85,B 0,C 180,E1 -11606.89,E2 -11606.89} C_VEL
LIN {X 0,Y 388.7,Z 629.5,A -85,B 0,C 180,E1 -11608.964,E2 -11608.964} C_VEL
LIN {X 0,Y 388.7,Z 629.499,A -85,B 0,C 180,E1 -11611.036,E2 -11611.036} C_VEL
LIN {X 0,Y 388.614,Z 628.318,A -85,B 0,C 180,E1 -11613.11,E2 -11613.11} C_VEL
LIN {X 0,Y 388.659,Z 625.984,A -85,B 0,C 180,E1 -11615.187,E2 -11615.187} C_VEL
LIN {X 0,Y 388.814,Z 622.448,A -85,B 0,C 180,E1 -11617.269,E2 -11617.269} C_VEL
LIN {X 0,Y 389.04,Z 617.616,A -85,B 0,C 180,E1 -11619.357,E2 -11619.357} C_VEL
LIN {X 0,Y 389.598,Z 611.365,A -85,B 0,C 180,E1 -11621.445,E2 -11621.445} C_VEL
LIN {X 0,Y 390.267,Z 603.514,A -85,B 0,C 180,E1 -11623.539,E2 -11623.539} C_VEL
LIN {X 0,Y 391.271,Z 595.174,A -85,B 0,C 180,E1 -11625.363,E2 -11625.363} C_VEL
LIN {X 0,Y 392.474,Z 585.128,A -85,B 0,C 180,E1 -11627.185,E2 -11627.185} C_VEL
LIN {X 0,Y 393.877,Z 574.106,A -85,B 0,C 180,E1 -11628.843,E2 -11628.843} C_VEL
LIN {X 0,Y 395.425,Z 561.473,A -85,B 0,C 180,E1 -11630.413,E2 -11630.413} C_VEL
LIN {X 0,Y 396.986,Z 549.013,A -85,B 0,C 180,E1 -11631.688,E2 -11631.688} C_VEL
LIN {X 0,Y 398.514,Z 535.367,A -85,B 0,C 180,E1 -11632.828,E2 -11632.828} C_VEL
LIN {X 0,Y 399.893,Z 521.235,A -85,B 0,C 180,E1 -11633.773,E2 -11633.773} C_VEL
LIN {X 0,Y 401.114,Z 505.717,A -85,B 0,C 180,E1 -11634.566,E2 -11634.566} C_VEL
LIN {X 0,Y 402.076,Z 490.752,A -85,B 0,C 180,E1 -11635.113,E2 -11635.113} C_VEL
LIN {X 0,Y 402.649,Z 474.783,A -85,B 0,C 180,E1 -11635.49,E2 -11635.49} C_VEL
LIN {X 0,Y 405.121,Z 355.556,A -85,B 0,C 180,E1 -11637.633,E2 -11637.633} C_VEL
LIN {X 0,Y 400.711,Z 331.641,A -85,B 0,C 180,E1 -11638.436,E2 -11638.436} C_VEL
LIN {X 0,Y 398.129,Z 320.117,A -85,B 0,C 180,E1 -11638.868,E2 -11638.868} C_VEL
LIN {X 0,Y 396.891,Z 316.806,A -85,B 0,C 180,E1 -11639.07,E2 -11639.07} C_VEL
LIN {X 0,Y 393.835,Z 303.863,A -85,B 0,C 180,E1 -11641.763,E2 -11641.763} C_VEL
LIN {X 0,Y 390.072,Z 289.542,A -85,B 0,C 180,E1 -11644.913,E2 -11644.913} C_VEL
LIN {X 0,Y 390.031,Z 289.528,A -85,B 0,C 180,E1 -11647.78,E2 -11647.78} C_VEL
LIN {X 0,Y 390.01,Z 289.53,A -85,B 0,C 180,E1 -11650.814,E2 -11650.814} C_VEL
LIN {X 0,Y 390.044,Z 289.527,A -85,B 0,C 180,E1 -11653.885,E2 -11653.885} C_VEL
LIN {X 0,Y 390.045,Z 289.523,A -85,B 0,C 180,E1 -11656.788,E2 -11656.788} C_VEL
LIN {X 0,Y 390.002,Z 289.529,A -85,B 0,C 180,E1 -11659.554,E2 -11659.554} C_VEL
LIN {X 0,Y 390.029,Z 289.525,A -85,B 0,C 180,E1 -11662.45,E2 -11662.45} C_VEL
LIN {X 0,Y 390.053,Z 289.523,A -85,B 0,C 180,E1 -11666.044,E2 -11666.044} C_VEL
LIN {X 0,Y 390.034,Z 289.523,A -85,B 0,C 180,E1 -11669.869,E2 -11669.869} C_VEL
LIN {X 0,Y 390.033,Z 289.521,A -85,B 0,C 180,E1 -11673.226,E2 -11673.226} C_VEL
LIN {X 0,Y 390.049,Z 289.52,A -85,B 0,C 180,E1 -11676.766,E2 -11676.766} C_VEL
LIN {X 0,Y 390.093,Z 289.502,A -85,B 0,C 180,E1 -11679.983,E2 -11679.983} C_VEL
LIN {X 0,Y 390.127,Z 289.507,A -85,B 0,C 180,E1 -11683.248,E2 -11683.248} C_VEL
LIN {X 0,Y 390.184,Z 289.498,A -85,B 0,C 180,E1 -11686.561,E2 -11686.561} C_VEL
LIN {X 0,Y 390.172,Z 289.5,A -85,B 0,C 180,E1 -11690.671,E2 -11690.671} C_VEL
LIN {X 0,Y 390.286,Z 289.488,A -85,B 0,C 180,E1 -11693.798,E2 -11693.798} C_VEL
LIN {X 0,Y 390.395,Z 289.474,A -85,B 0,C 180,E1 -11697.937,E2 -11697.937} C_VEL
LIN {X 0,Y 390.399,Z 289.474,A -85,B 0,C 180,E1 -11702.063,E2 -11702.063} C_VEL
LIN {X 0,Y 390.267,Z 289.49,A -85,B 0,C 180,E1 -11706.587,E2 -11706.587} C_VEL
LIN {X 0,Y 390.181,Z 289.508,A -85,B 0,C 180,E1 -11709.329,E2 -11709.329} C_VEL
LIN {X 0,Y 390.159,Z 289.507,A -85,B 0,C 180,E1 -11712.484,E2 -11712.484} C_VEL
LIN {X 0,Y 390.127,Z 289.513,A -85,B 0,C 180,E1 -11715.677,E2 -11715.677} C_VEL
LIN {X 0,Y 390.092,Z 289.508,A -85,B 0,C 180,E1 -11718.923,E2 -11718.923} C_VEL
LIN {X 0,Y 390.029,Z 289.516,A -85,B 0,C 180,E1 -11722.235,E2 -11722.235} C_VEL
LIN {X 0,Y 390.088,Z 289.511,A -85,B 0,C 180,E1 -11725.737,E2 -11725.737} C_VEL
LIN {X 0,Y 390.087,Z 289.504,A -85,B 0,C 180,E1 -11728.02,E2 -11728.02} C_VEL
LIN {X 0,Y 390.014,Z 289.524,A -85,B 0,C 180,E1 -11731.505,E2 -11731.505} C_VEL
LIN {X 0,Y 390.062,Z 289.521,A -85,B 0,C 180,E1 -11735.209,E2 -11735.209} C_VEL
LIN {X 0,Y 390.081,Z 289.519,A -85,B 0,C 180,E1 -11739.094,E2 -11739.094} C_VEL
LIN {X 0,Y 390.036,Z 289.524,A -85,B 0,C 180,E1 -11742.375,E2 -11742.375} C_VEL
LIN {X 0,Y 390.039,Z 289.525,A -85,B 0,C 180,E1 -11745.355,E2 -11745.355} C_VEL
LIN {X 0,Y 390.027,Z 289.528,A -85,B 0,C 180,E1 -11748.188,E2 -11748.188} C_VEL
LIN {X 0,Y 390.087,Z 289.512,A -85,B 0,C 180,E1 -11750.909,E2 -11750.909} C_VEL
LIN {X 0,Y 390.081,Z 289.516,A -85,B 0,C 180,E1 -11754.794,E2 -11754.794} C_VEL
LIN {X 0,Y 390.068,Z 289.624,A -85,B 0,C 180,E1 -11758.652,E2 -11758.652} C_VEL
LIN {X 0,Y 392.255,Z 298.029,A -85,B 0,C 180,E1 -11760.655,E2 -11760.655} C_VEL
LIN {X 0,Y 401.264,Z 317.663,A -85,B 0,C 180,E1 -11761.775,E2 -11761.775} C_VEL
LIN {X 0,Y 405.376,Z 327.958,A -85,B 0,C 180,E1 -11762.292,E2 -11762.292} C_VEL
LIN {X 0,Y 405.492,Z 333.072,A -85,B 0,C 180,E1 -11762.401,E2 -11762.401} C_VEL
LIN {X 0,Y 403.203,Z 440.941,A -85,B 0,C 180,E1 -11764.34,E2 -11764.34} C_VEL
LIN {X 0,Y 402.616,Z 465.014,A -85,B 0,C 180,E1 -11764.819,E2 -11764.819} C_VEL
LIN {X 0,Y 401.903,Z 479.846,A -85,B 0,C 180,E1 -11765.304,E2 -11765.304} C_VEL
LIN {X 0,Y 401.149,Z 492.332,A -85,B 0,C 180,E1 -11765.873,E2 -11765.873} C_VEL
LIN {X 0,Y 399.991,Z 506.597,A -85,B 0,C 180,E1 -11766.714,E2 -11766.714} C_VEL
LIN {X 0,Y 398.589,Z 520.174,A -85,B 0,C 180,E1 -11767.723,E2 -11767.723} C_VEL
LIN {X 0,Y 397.056,Z 533.943,A -85,B 0,C 180,E1 -11768.997,E2 -11768.997} C_VEL
LIN {X 0,Y 395.554,Z 546.398,A -85,B 0,C 180,E1 -11770.411,E2 -11770.411} C_VEL
LIN {X 0,Y 394.211,Z 556.754,A -85,B 0,C 180,E1 -11771.821,E2 -11771.821} C_VEL
LIN {X 0,Y 392.956,Z 566.393,A -85,B 0,C 180,E1 -11773.372,E2 -11773.372} C_VEL
LIN {X 0,Y 391.732,Z 575.838,A -85,B 0,C 180,E1 -11775.188,E2 -11775.188} C_VEL
LIN {X 0,Y 390.832,Z 583.696,A -85,B 0,C 180,E1 -11777.011,E2 -11777.011} C_VEL
LIN {X 0,Y 389.924,Z 591.033,A -85,B 0,C 180,E1 -11779.091,E2 -11779.091} C_VEL
LIN {X 0,Y 389.393,Z 596.85,A -85,B 0,C 180,E1 -11781.175,E2 -11781.175} C_VEL
LIN {X 0,Y 389.126,Z 600.293,A -85,B 0,C 180,E1 -11782.737,E2 -11782.737} C_VEL
LIN {X 0,Y 388.889,Z 603.782,A -85,B 0,C 180,E1 -11784.816,E2 -11784.816} C_VEL
LIN {X 0,Y 388.726,Z 606.091,A -85,B 0,C 180,E1 -11786.891,E2 -11786.891} C_VEL
LIN {X 0,Y 388.716,Z 607.131,A -85,B 0,C 180,E1 -11788.649,E2 -11788.649} C_VEL
LIN {X 0,Y 388.057,Z 607.43,A -85,B 0,C 180,E1 -11789.514,E2 -11789.514} C_VEL
LIN {X 0,Y 385.186,Z 607.521,A -85,B 0,C 180,E1 -11790.92,E2 -11790.92} C_VEL
LIN {X 0,Y 382.752,Z 607.154,A -85,B 0,C 180,E1 -11792.055,E2 -11792.055} C_VEL
LIN {X 0,Y 381.709,Z 606.575,A -85,B 0,C 180,E1 -11792.93,E2 -11792.93} C_VEL
LIN {X 0,Y 381.626,Z 606.318,A -85,B 0,C 180,E1 -11793.225,E2 -11793.225} C_VEL
LIN {X 0,Y 381.804,Z 604.124,A -85,B 0,C 180,E1 -11795.281,E2 -11795.281} C_VEL
LIN {X 0,Y 382.037,Z 600.693,A -85,B 0,C 180,E1 -11797.398,E2 -11797.398} C_VEL
LIN {X 0,Y 382.45,Z 595.993,A -85,B 0,C 180,E1 -11799.519,E2 -11799.519} C_VEL
LIN {X 0,Y 383.081,Z 589.902,A -85,B 0,C 180,E1 -11801.642,E2 -11801.642} C_VEL
LIN {X 0,Y 383.931,Z 583.278,A -85,B 0,C 180,E1 -11803.497,E2 -11803.497} C_VEL
LIN {X 0,Y 385.098,Z 574.043,A -85,B 0,C 180,E1 -11805.615,E2 -11805.615} C_VEL
LIN {X 0,Y 386.489,Z 564.179,A -85,B 0,C 180,E1 -11807.459,E2 -11807.459} C_VEL
LIN {X 0,Y 388.067,Z 552.852,A -85,B 0,C 180,E1 -11809.206,E2 -11809.206} C_VEL
LIN {X 0,Y 389.592,Z 540.912,A -85,B 0,C 180,E1 -11810.733,E2 -11810.733} C_VEL
LIN {X 0,Y 391.202,Z 528.636,A -85,B 0,C 180,E1 -11812.025,E2 -11812.025} C_VEL
LIN {X 0,Y 392.682,Z 515.216,A -85,B 0,C 180,E1 -11813.187,E2 -11813.187} C_VEL
LIN {X 0,Y 394.093,Z 500.26,A -85,B 0,C 180,E1 -11814.215,E2 -11814.215} C_VEL
LIN {X 0,Y 395.148,Z 485.465,A -85,B 0,C 180,E1 -11814.997,E2 -11814.997} C_VEL
LIN {X 0,Y 396.04,Z 469.63,A -85,B 0,C 180,E1 -11815.594,E2 -11815.594} C_VEL
LIN {X 0,Y 396.677,Z 453.435,A -85,B 0,C 180,E1 -11815.972,E2 -11815.972} C_VEL
LIN {X 0,Y 399.262,Z 329.742,A -85,B 0,C 180,E1 -11818.241,E2 -11818.241} C_VEL
LIN {X 0,Y 390.856,Z 310.449,A -85,B 0,C 180,E1 -11819.308,E2 -11819.308} C_VEL
LIN {X 0,Y 384.989,Z 298.051,A -85,B 0,C 180,E1 -11820.08,E2 -11820.08} C_VEL
LIN {X 0,Y 382.988,Z 290.405,A -85,B 0,C 180,E1 -11821.996,E2 -11821.996} C_VEL
LIN {X 0,Y 383.016,Z 290.4,A -85,B 0,C 180,E1 -11824.667,E2 -11824.667} C_VEL
LIN {X 0,Y 382.997,Z 290.404,A -85,B 0,C 180,E1 -11827.903,E2 -11827.903} C_VEL
LIN {X 0,Y 382.98,Z 290.402,A -85,B 0,C 180,E1 -11831.347,E2 -11831.347} C_VEL
LIN {X 0,Y 382.991,Z 290.402,A -85,B 0,C 180,E1 -11834.302,E2 -11834.302} C_VEL
LIN {X 0,Y 383.005,Z 290.393,A -85,B 0,C 180,E1 -11837.239,E2 -11837.239} C_VEL
LIN {X 0,Y 383.004,Z 290.4,A -85,B 0,C 180,E1 -11840.414,E2 -11840.414} C_VEL
LIN {X 0,Y 383.008,Z 290.389,A -85,B 0,C 180,E1 -11844.042,E2 -11844.042} C_VEL
LIN {X 0,Y 382.977,Z 290.397,A -85,B 0,C 180,E1 -11847.578,E2 -11847.578} C_VEL
LIN {X 0,Y 382.98,Z 290.389,A -85,B 0,C 180,E1 -11850.299,E2 -11850.299} C_VEL
LIN {X 0,Y 383.041,Z 290.391,A -85,B 0,C 180,E1 -11853.874,E2 -11853.874} C_VEL
LIN {X 0,Y 382.981,Z 290.4,A -85,B 0,C 180,E1 -11857.333,E2 -11857.333} C_VEL
LIN {X 0,Y 383.048,Z 290.398,A -85,B 0,C 180,E1 -11860.716,E2 -11860.716} C_VEL
LIN {X 0,Y 383.069,Z 290.391,A -85,B 0,C 180,E1 -11864.026,E2 -11864.026} C_VEL
LIN {X 0,Y 383.125,Z 290.384,A -85,B 0,C 180,E1 -11867.283,E2 -11867.283} C_VEL
LIN {X 0,Y 383.131,Z 290.382,A -85,B 0,C 180,E1 -11870.497,E2 -11870.497} C_VEL
LIN {X 0,Y 383.249,Z 290.368,A -85,B 0,C 180,E1 -11873.683,E2 -11873.683} C_VEL
LIN {X 0,Y 383.368,Z 290.354,A -85,B 0,C 180,E1 -11877.899,E2 -11877.899} C_VEL
LIN {X 0,Y 383.501,Z 290.332,A -85,B 0,C 180,E1 -11880,E2 -11880} C_VEL
LIN {X 0,Y 383.19,Z 290.375,A -85,B 0,C 180,E1 -11883.154,E2 -11883.154} C_VEL
LIN {X 0,Y 383.248,Z 290.37,A -85,B 0,C 180,E1 -11886.317,E2 -11886.317} C_VEL
LIN {X 0,Y 383.128,Z 290.379,A -85,B 0,C 180,E1 -11889.503,E2 -11889.503} C_VEL
LIN {X 0,Y 383.115,Z 290.379,A -85,B 0,C 180,E1 -11893.536,E2 -11893.536} C_VEL
LIN {X 0,Y 383.083,Z 290.387,A -85,B 0,C 180,E1 -11897.07,E2 -11897.07} C_VEL
LIN {X 0,Y 383.018,Z 290.399,A -85,B 0,C 180,E1 -11900.647,E2 -11900.647} C_VEL
LIN {X 0,Y 382.998,Z 290.403,A -85,B 0,C 180,E1 -11903.81,E2 -11903.81} C_VEL
LIN {X 0,Y 382.978,Z 290.403,A -85,B 0,C 180,E1 -11907.308,E2 -11907.308} C_VEL
LIN {X 0,Y 382.973,Z 290.404,A -85,B 0,C 180,E1 -11910.919,E2 -11910.919} C_VEL
LIN {X 0,Y 383.002,Z 290.402,A -85,B 0,C 180,E1 -11914.669,E2 -11914.669} C_VEL
LIN {X 0,Y 382.983,Z 290.405,A -85,B 0,C 180,E1 -11917.903,E2 -11917.903} C_VEL
LIN {X 0,Y 382.954,Z 290.393,A -85,B 0,C 180,E1 -11921.351,E2 -11921.351} C_VEL
LIN {X 0,Y 382.986,Z 290.402,A -85,B 0,C 180,E1 -11924.303,E2 -11924.303} C_VEL
LIN {X 0,Y 382.976,Z 290.404,A -85,B 0,C 180,E1 -11927.237,E2 -11927.237} C_VEL
LIN {X 0,Y 382.979,Z 290.403,A -85,B 0,C 180,E1 -11930.42,E2 -11930.42} C_VEL
LIN {X 0,Y 383.018,Z 290.4,A -85,B 0,C 180,E1 -11934.045,E2 -11934.045} C_VEL
LIN {X 0,Y 383.056,Z 290.493,A -85,B 0,C 180,E1 -11934.575,E2 -11934.575} C_VEL
LIN {X 0,Y 386.552,Z 303.709,A -85,B 0,C 180,E1 -11937.566,E2 -11937.566} C_VEL
LIN {X 0,Y 389.734,Z 317.094,A -85,B 0,C 180,E1 -11940.38,E2 -11940.38} C_VEL
LIN {X 0,Y 392.73,Z 324.482,A -85,B 0,C 180,E1 -11940.778,E2 -11940.778} C_VEL
LIN {X 0,Y 398.437,Z 353.681,A -85,B 0,C 180,E1 -11941.818,E2 -11941.818} C_VEL
LIN {X 0,Y 398.837,Z 357.134,A -85,B 0,C 180,E1 -11941.917,E2 -11941.917} C_VEL
LIN {X 0,Y 396.045,Z 482.748,A -85,B 0,C 180,E1 -11944.231,E2 -11944.231} C_VEL
LIN {X 0,Y 395.221,Z 498.242,A -85,B 0,C 180,E1 -11944.702,E2 -11944.702} C_VEL
LIN {X 0,Y 394.112,Z 512.861,A -85,B 0,C 180,E1 -11945.348,E2 -11945.348} C_VEL
LIN {X 0,Y 392.889,Z 526.187,A -85,B 0,C 180,E1 -11946.127,E2 -11946.127} C_VEL
LIN {X 0,Y 391.373,Z 540.085,A -85,B 0,C 180,E1 -11947.15,E2 -11947.15} C_VEL
LIN {X 0,Y 389.854,Z 552.823,A -85,B 0,C 180,E1 -11948.312,E2 -11948.312} C_VEL
LIN {X 0,Y 388.154,Z 565.708,A -85,B 0,C 180,E1 -11949.741,E2 -11949.741} C_VEL
LIN {X 0,Y 386.806,Z 576.505,A -85,B 0,C 180,E1 -11951.186,E2 -11951.186} C_VEL
LIN {X 0,Y 385.417,Z 586.494,A -85,B 0,C 180,E1 -11952.764,E2 -11952.764} C_VEL
LIN {X 0,Y 384.174,Z 596.273,A -85,B 0,C 180,E1 -11954.618,E2 -11954.618} C_VEL
LIN {X 0,Y 383.187,Z 604.242,A -85,B 0,C 180,E1 -11956.426,E2 -11956.426} C_VEL
LIN {X 0,Y 382.581,Z 611.19,A -85,B 0,C 180,E1 -11958.342,E2 -11958.342} C_VEL
LIN {X 0,Y 381.983,Z 617.428,A -85,B 0,C 180,E1 -11960.469,E2 -11960.469} C_VEL
LIN {X 0,Y 381.732,Z 622.257,A -85,B 0,C 180,E1 -11962.596,E2 -11962.596} C_VEL
LIN {X 0,Y 381.584,Z 625.796,A -85,B 0,C 180,E1 -11964.716,E2 -11964.716} C_VEL
LIN {X 0,Y 381.526,Z 628.124,A -85,B 0,C 180,E1 -11966.832,E2 -11966.832} C_VEL
LIN {X 0,Y 381.614,Z 629.298,A -85,B 0,C 180,E1 -11968.945,E2 -11968.945} C_VEL
LIN {X 0,Y 381.614,Z 629.296,A -85,B 0,C 180,E1 -11971.055,E2 -11971.055} C_VEL
LIN {X 0,Y 381.525,Z 628.114,A -85,B 0,C 180,E1 -11973.168,E2 -11973.168} C_VEL
LIN {X 0,Y 381.572,Z 625.781,A -85,B 0,C 180,E1 -11975.284,E2 -11975.284} C_VEL
LIN {X 0,Y 381.719,Z 622.243,A -85,B 0,C 180,E1 -11977.405,E2 -11977.405} C_VEL
LIN {X 0,Y 381.982,Z 617.41,A -85,B 0,C 180,E1 -11979.531,E2 -11979.531} C_VEL
LIN {X 0,Y 382.58,Z 611.159,A -85,B 0,C 180,E1 -11981.658,E2 -11981.658} C_VEL
LIN {X 0,Y 383.318,Z 603.308,A -85,B 0,C 180,E1 -11983.789,E2 -11983.789} C_VEL
LIN {X 0,Y 384.355,Z 594.967,A -85,B 0,C 180,E1 -11985.646,E2 -11985.646} C_VEL
LIN {X 0,Y 385.642,Z 584.921,A -85,B 0,C 180,E1 -11987.499,E2 -11987.499} C_VEL
LIN {X 0,Y 386.999,Z 574.651,A -85,B 0,C 180,E1 -11989.079,E2 -11989.079} C_VEL
LIN {X 0,Y 388.566,Z 562.417,A -85,B 0,C 180,E1 -11990.652,E2 -11990.652} C_VEL
LIN {X 0,Y 390.2,Z 550.145,A -85,B 0,C 180,E1 -11991.945,E2 -11991.945} C_VEL
LIN {X 0,Y 391.779,Z 536.791,A -85,B 0,C 180,E1 -11993.104,E2 -11993.104} C_VEL
LIN {X 0,Y 393.282,Z 522.053,A -85,B 0,C 180,E1 -11994.127,E2 -11994.127} C_VEL
LIN {X 0,Y 394.542,Z 507.143,A -85,B 0,C 180,E1 -11994.922,E2 -11994.922} C_VEL
LIN {X 0,Y 395.53,Z 492.478,A -85,B 0,C 180,E1 -11995.488,E2 -11995.488} C_VEL
LIN {X 0,Y 396.14,Z 477.766,A -85,B 0,C 180,E1 -11995.869,E2 -11995.869} C_VEL
LIN {X 0,Y 398.735,Z 359.857,A -85,B 0,C 180,E1 -11998.025,E2 -11998.025} C_VEL
LIN {X 0,Y 398.6,Z 355.125,A -85,B 0,C 180,E1 -11998.129,E2 -11998.129} C_VEL
LIN {X 0,Y 393.963,Z 330.552,A -85,B 0,C 180,E1 -11998.987,E2 -11998.987} C_VEL
LIN {X 0,Y 392.076,Z 322.554,A -85,B 0,C 180,E1 -11999.302,E2 -11999.302} C_VEL
LIN {X 0,Y 389.655,Z 316.696,A -85,B 0,C 180,E1 -11999.64,E2 -11999.64} C_VEL
LIN {X 0,Y 386.524,Z 303.628,A -85,B 0,C 180,E1 -12002.437,E2 -12002.437} C_VEL
LIN {X 0,Y 383.027,Z 290.398,A -85,B 0,C 180,E1 -12005.469,E2 -12005.469} C_VEL
LIN {X 0,Y 382.975,Z 290.408,A -85,B 0,C 180,E1 -12008.603,E2 -12008.603} C_VEL
LIN {X 0,Y 382.954,Z 290.408,A -85,B 0,C 180,E1 -12011.35,E2 -12011.35} C_VEL
LIN {X 0,Y 382.986,Z 290.406,A -85,B 0,C 180,E1 -12014.302,E2 -12014.302} C_VEL
LIN {X 0,Y 383.004,Z 290.4,A -85,B 0,C 180,E1 -12017.239,E2 -12017.239} C_VEL
LIN {X 0,Y 382.977,Z 290.405,A -85,B 0,C 180,E1 -12020.418,E2 -12020.418} C_VEL
LIN {X 0,Y 383.004,Z 290.399,A -85,B 0,C 180,E1 -12024.042,E2 -12024.042} C_VEL
LIN {X 0,Y 382.976,Z 290.401,A -85,B 0,C 180,E1 -12027.578,E2 -12027.578} C_VEL
LIN {X 0,Y 382.968,Z 290.404,A -85,B 0,C 180,E1 -12030.298,E2 -12030.298} C_VEL
LIN {X 0,Y 382.994,Z 290.404,A -85,B 0,C 180,E1 -12034.044,E2 -12034.044} C_VEL
LIN {X 0,Y 382.976,Z 290.404,A -85,B 0,C 180,E1 -12037.333,E2 -12037.333} C_VEL
LIN {X 0,Y 383.047,Z 290.375,A -85,B 0,C 180,E1 -12040.716,E2 -12040.716} C_VEL
LIN {X 0,Y 383.068,Z 290.393,A -85,B 0,C 180,E1 -12044.026,E2 -12044.026} C_VEL
LIN {X 0,Y 383.122,Z 290.368,A -85,B 0,C 180,E1 -12047.284,E2 -12047.284} C_VEL
LIN {X 0,Y 383.123,Z 290.378,A -85,B 0,C 180,E1 -12050.497,E2 -12050.497} C_VEL
LIN {X 0,Y 383.243,Z 290.367,A -85,B 0,C 180,E1 -12053.683,E2 -12053.683} C_VEL
LIN {X 0,Y 383.361,Z 290.35,A -85,B 0,C 180,E1 -12057.899,E2 -12057.899} C_VEL
LIN {X 0,Y 383.365,Z 290.35,A -85,B 0,C 180,E1 -12062.101,E2 -12062.101} C_VEL
LIN {X 0,Y 383.228,Z 290.367,A -85,B 0,C 180,E1 -12066.578,E2 -12066.578} C_VEL
LIN {X 0,Y 383.131,Z 290.384,A -85,B 0,C 180,E1 -12069.503,E2 -12069.503} C_VEL
LIN {X 0,Y 383.116,Z 290.386,A -85,B 0,C 180,E1 -12073.536,E2 -12073.536} C_VEL
LIN {X 0,Y 383.084,Z 290.394,A -85,B 0,C 180,E1 -12077.07,E2 -12077.07} C_VEL
LIN {X 0,Y 383.019,Z 290.376,A -85,B 0,C 180,E1 -12080.647,E2 -12080.647} C_VEL
LIN {X 0,Y 383.013,Z 290.399,A -85,B 0,C 180,E1 -12083.809,E2 -12083.809} C_VEL
LIN {X 0,Y 383.046,Z 290.377,A -85,B 0,C 180,E1 -12087.303,E2 -12087.303} C_VEL
LIN {X 0,Y 382.974,Z 290.407,A -85,B 0,C 180,E1 -12090.919,E2 -12090.919} C_VEL
LIN {X 0,Y 383.004,Z 290.4,A -85,B 0,C 180,E1 -12094.67,E2 -12094.67} C_VEL
LIN {X 0,Y 382.991,Z 290.398,A -85,B 0,C 180,E1 -12097.904,E2 -12097.904} C_VEL
LIN {X 0,Y 382.977,Z 290.403,A -85,B 0,C 180,E1 -12101.348,E2 -12101.348} C_VEL
LIN {X 0,Y 382.99,Z 290.403,A -85,B 0,C 180,E1 -12104.304,E2 -12104.304} C_VEL
LIN {X 0,Y 383.006,Z 290.403,A -85,B 0,C 180,E1 -12107.241,E2 -12107.241} C_VEL
LIN {X 0,Y 383.012,Z 290.398,A -85,B 0,C 180,E1 -12110.414,E2 -12110.414} C_VEL
LIN {X 0,Y 383.021,Z 290.393,A -85,B 0,C 180,E1 -12114.045,E2 -12114.045} C_VEL
LIN {X 0,Y 382.984,Z 290.405,A -85,B 0,C 180,E1 -12117.579,E2 -12117.579} C_VEL
LIN {X 0,Y 383.015,Z 290.53,A -85,B 0,C 180,E1 -12118.162,E2 -12118.162} C_VEL
LIN {X 0,Y 385.103,Z 298.421,A -85,B 0,C 180,E1 -12120.058,E2 -12120.058} C_VEL
LIN {X 0,Y 394.683,Z 318.813,A -85,B 0,C 180,E1 -12121.279,E2 -12121.279} C_VEL
LIN {X 0,Y 399.233,Z 329.846,A -85,B 0,C 180,E1 -12121.861,E2 -12121.861} C_VEL
LIN {X 0,Y 397.072,Z 432.235,A -85,B 0,C 180,E1 -12123.738,E2 -12123.738} C_VEL
LIN {X 0,Y 396.234,Z 464.095,A -85,B 0,C 180,E1 -12124.349,E2 -12124.349} C_VEL
LIN {X 0,Y 395.562,Z 479.281,A -85,B 0,C 180,E1 -12124.845,E2 -12124.845} C_VEL
LIN {X 0,Y 394.644,Z 493.065,A -85,B 0,C 180,E1 -12125.477,E2 -12125.477} C_VEL
LIN {X 0,Y 393.487,Z 506.807,A -85,B 0,C 180,E1 -12126.306,E2 -12126.306} C_VEL
LIN {X 0,Y 392.011,Z 520.383,A -85,B 0,C 180,E1 -12127.329,E2 -12127.329} C_VEL
LIN {X 0,Y 390.444,Z 534.15,A -85,B 0,C 180,E1 -12128.624,E2 -12128.624} C_VEL
LIN {X 0,Y 388.874,Z 546.257,A -85,B 0,C 180,E1 -12130.015,E2 -12130.015} C_VEL
LIN {X 0,Y 387.445,Z 556.961,A -85,B 0,C 180,E1 -12131.492,E2 -12131.492} C_VEL
LIN {X 0,Y 386.126,Z 566.6,A -85,B 0,C 180,E1 -12133.069,E2 -12133.069} C_VEL
LIN {X 0,Y 384.838,Z 576.044,A -85,B 0,C 180,E1 -12134.916,E2 -12134.916} C_VEL
LIN {X 0,Y 383.874,Z 583.902,A -85,B 0,C 180,E1 -12136.771,E2 -12136.771} C_VEL
LIN {X 0,Y 382.926,Z 591.238,A -85,B 0,C 180,E1 -12138.889,E2 -12138.889} C_VEL
LIN {X 0,Y 382.358,Z 597.055,A -85,B 0,C 180,E1 -12141.012,E2 -12141.012} C_VEL
LIN {X 0,Y 382.058,Z 600.498,A -85,B 0,C 180,E1 -12142.602,E2 -12142.602} C_VEL
LIN {X 0,Y 381.812,Z 603.986,A -85,B 0,C 180,E1 -12144.719,E2 -12144.719} C_VEL
LIN {X 0,Y 381.632,Z 606.294,A -85,B 0,C 180,E1 -12146.833,E2 -12146.833} C_VEL
LIN {X 0,Y 381.64,Z 607.471,A -85,B 0,C 180,E1 -12148.945,E2 -12148.945} C_VEL
LIN {X 0,Y 381.641,Z 607.486,A -85,B 0,C 180,E1 -12151.055,E2 -12151.055} C_VEL
LIN {X 0,Y 381.626,Z 606.318,A -85,B 0,C 180,E1 -12153.225,E2 -12153.225} C_VEL
LIN {X 0,Y 380.98,Z 605.563,A -85,B 0,C 180,E1 -12154.098,E2 -12154.098} C_VEL
LIN {X 0,Y 378.222,Z 603.977,A -85,B 0,C 180,E1 -12155.517,E2 -12155.517} C_VEL
LIN {X 0,Y 375.947,Z 602.391,A -85,B 0,C 180,E1 -12156.654,E2 -12156.654} C_VEL
LIN {X 0,Y 375.05,Z 600.931,A -85,B 0,C 180,E1 -12157.521,E2 -12157.521} C_VEL
LIN {X 0,Y 375.02,Z 600.361,A -85,B 0,C 180,E1 -12157.812,E2 -12157.812} C_VEL
LIN {X 0,Y 375.424,Z 596.195,A -85,B 0,C 180,E1 -12159.699,E2 -12159.699} C_VEL
LIN {X 0,Y 376.11,Z 590.104,A -85,B 0,C 180,E1 -12161.861,E2 -12161.861} C_VEL
LIN {X 0,Y 376.963,Z 583.481,A -85,B 0,C 180,E1 -12163.751,E2 -12163.751} C_VEL
LIN {X 0,Y 378.046,Z 575.475,A -85,B 0,C 180,E1 -12165.638,E2 -12165.638} C_VEL
LIN {X 0,Y 379.449,Z 565.865,A -85,B 0,C 180,E1 -12167.516,E2 -12167.516} C_VEL
LIN {X 0,Y 380.899,Z 556.035,A -85,B 0,C 180,E1 -12169.117,E2 -12169.117} C_VEL
LIN {X 0,Y 382.379,Z 545.406,A -85,B 0,C 180,E1 -12170.579,E2 -12170.579} C_VEL
LIN {X 0,Y 383.93,Z 533.984,A -85,B 0,C 180,E1 -12171.898,E2 -12171.898} C_VEL
LIN {X 0,Y 385.393,Z 521.72,A -85,B 0,C 180,E1 -12173.083,E2 -12173.083} C_VEL
LIN {X 0,Y 386.906,Z 508.4,A -85,B 0,C 180,E1 -12174.123,E2 -12174.123} C_VEL
LIN {X 0,Y 388.236,Z 493.513,A -85,B 0,C 180,E1 -12175.043,E2 -12175.043} C_VEL
LIN {X 0,Y 389.183,Z 479.054,A -85,B 0,C 180,E1 -12175.719,E2 -12175.719} C_VEL
LIN {X 0,Y 389.949,Z 464.125,A -85,B 0,C 180,E1 -12176.203,E2 -12176.203} C_VEL
LIN {X 0,Y 391.207,Z 416.084,A -85,B 0,C 180,E1 -12177.119,E2 -12177.119} C_VEL
LIN {X 0,Y 393.034,Z 331.753,A -85,B 0,C 180,E1 -12178.692,E2 -12178.692} C_VEL
LIN {X 0,Y 384.435,Z 312.045,A -85,B 0,C 180,E1 -12179.816,E2 -12179.816} C_VEL
LIN {X 0,Y 377.781,Z 298.29,A -85,B 0,C 180,E1 -12180.713,E2 -12180.713} C_VEL
LIN {X 0,Y 375.948,Z 291.282,A -85,B 0,C 180,E1 -12182.509,E2 -12182.509} C_VEL
LIN {X 0,Y 375.955,Z 291.285,A -85,B 0,C 180,E1 -12185.415,E2 -12185.415} C_VEL
LIN {X 0,Y 375.971,Z 291.281,A -85,B 0,C 180,E1 -12188.27,E2 -12188.27} C_VEL
LIN {X 0,Y 375.93,Z 291.284,A -85,B 0,C 180,E1 -12191.6,E2 -12191.6} C_VEL
LIN {X 0,Y 375.921,Z 291.284,A -85,B 0,C 180,E1 -12195.268,E2 -12195.268} C_VEL
LIN {X 0,Y 375.926,Z 291.267,A -85,B 0,C 180,E1 -12198.399,E2 -12198.399} C_VEL
LIN {X 0,Y 375.964,Z 291.272,A -85,B 0,C 180,E1 -12201.73,E2 -12201.73} C_VEL
LIN {X 0,Y 375.967,Z 291.276,A -85,B 0,C 180,E1 -12205.333,E2 -12205.333} C_VEL
LIN {X 0,Y 375.948,Z 291.265,A -85,B 0,C 180,E1 -12208.437,E2 -12208.437} C_VEL
LIN {X 0,Y 375.973,Z 291.275,A -85,B 0,C 180,E1 -12212.139,E2 -12212.139} C_VEL
LIN {X 0,Y 375.983,Z 291.271,A -85,B 0,C 180,E1 -12214.537,E2 -12214.537} C_VEL
LIN {X 0,Y 375.947,Z 291.274,A -85,B 0,C 180,E1 -12218.045,E2 -12218.045} C_VEL
LIN {X 0,Y 375.993,Z 291.269,A -85,B 0,C 180,E1 -12221.472,E2 -12221.472} C_VEL
LIN {X 0,Y 376.047,Z 291.27,A -85,B 0,C 180,E1 -12224.832,E2 -12224.832} C_VEL
LIN {X 0,Y 376.037,Z 291.266,A -85,B 0,C 180,E1 -12228.136,E2 -12228.136} C_VEL
LIN {X 0,Y 376.189,Z 291.244,A -85,B 0,C 180,E1 -12231.941,E2 -12231.941} C_VEL
LIN {X 0,Y 376.146,Z 291.252,A -85,B 0,C 180,E1 -12234.639,E2 -12234.639} C_VEL
LIN {X 0,Y 376.333,Z 291.23,A -85,B 0,C 180,E1 -12237.859,E2 -12237.859} C_VEL
LIN {X 0,Y 376.471,Z 291.208,A -85,B 0,C 180,E1 -12240,E2 -12240} C_VEL
LIN {X 0,Y 376.327,Z 291.232,A -85,B 0,C 180,E1 -12242.14,E2 -12242.14} C_VEL
LIN {X 0,Y 376.206,Z 291.248,A -85,B 0,C 180,E1 -12246.436,E2 -12246.436} C_VEL
LIN {X 0,Y 376.099,Z 291.254,A -85,B 0,C 180,E1 -12249.682,E2 -12249.682} C_VEL
LIN {X 0,Y 376.08,Z 291.256,A -85,B 0,C 180,E1 -12253.658,E2 -12253.658} C_VEL
LIN {X 0,Y 376.022,Z 291.266,A -85,B 0,C 180,E1 -12257.4,E2 -12257.4} C_VEL
LIN {X 0,Y 375.969,Z 291.276,A -85,B 0,C 180,E1 -12260.832,E2 -12260.832} C_VEL
LIN {X 0,Y 375.948,Z 291.284,A -85,B 0,C 180,E1 -12264.284,E2 -12264.284} C_VEL
LIN {X 0,Y 375.922,Z 291.285,A -85,B 0,C 180,E1 -12267.865,E2 -12267.865} C_VEL
LIN {X 0,Y 375.948,Z 291.28,A -85,B 0,C 180,E1 -12271.563,E2 -12271.563} C_VEL
LIN {X 0,Y 375.94,Z 291.28,A -85,B 0,C 180,E1 -12275.417,E2 -12275.417} C_VEL
LIN {X 0,Y 375.926,Z 291.283,A -85,B 0,C 180,E1 -12278.263,E2 -12278.263} C_VEL
LIN {X 0,Y 375.91,Z 291.272,A -85,B 0,C 180,E1 -12281.598,E2 -12281.598} C_VEL
LIN {X 0,Y 375.916,Z 291.284,A -85,B 0,C 180,E1 -12284.731,E2 -12284.731} C_VEL
LIN {X 0,Y 375.901,Z 291.287,A -85,B 0,C 180,E1 -12287.697,E2 -12287.697} C_VEL
LIN {X 0,Y 375.928,Z 291.282,A -85,B 0,C 180,E1 -12290.534,E2 -12290.534} C_VEL
LIN {X 0,Y 376.013,Z 291.453,A -85,B 0,C 180,E1 -12294.056,E2 -12294.056} C_VEL
LIN {X 0,Y 379.448,Z 304.2,A -85,B 0,C 180,E1 -12297.026,E2 -12297.026} C_VEL
LIN {X 0,Y 382.396,Z 316.583,A -85,B 0,C 180,E1 -12299.746,E2 -12299.746} C_VEL
LIN {X 0,Y 386.873,Z 327.343,A -85,B 0,C 180,E1 -12300.355,E2 -12300.355} C_VEL
LIN {X 0,Y 392.523,Z 356.822,A -85,B 0,C 180,E1 -12301.422,E2 -12301.422} C_VEL
LIN {X 0,Y 390.303,Z 458.82,A -85,B 0,C 180,E1 -12303.319,E2 -12303.319} C_VEL
LIN {X 0,Y 389.535,Z 484.977,A -85,B 0,C 180,E1 -12303.839,E2 -12303.839} C_VEL
LIN {X 0,Y 388.593,Z 500.577,A -85,B 0,C 180,E1 -12304.354,E2 -12304.354} C_VEL
LIN {X 0,Y 387.432,Z 515.31,A -85,B 0,C 180,E1 -12305.053,E2 -12305.053} C_VEL
LIN {X 0,Y 385.963,Z 529.924,A -85,B 0,C 180,E1 -12305.969,E2 -12305.969} C_VEL
LIN {X 0,Y 384.444,Z 542.984,A -85,B 0,C 180,E1 -12306.999,E2 -12306.999} C_VEL
LIN {X 0,Y 382.675,Z 556.426,A -85,B 0,C 180,E1 -12308.309,E2 -12308.309} C_VEL
LIN {X 0,Y 380.983,Z 568.869,A -85,B 0,C 180,E1 -12309.793,E2 -12309.793} C_VEL
LIN {X 0,Y 379.554,Z 579.892,A -85,B 0,C 180,E1 -12311.378,E2 -12311.378} C_VEL
LIN {X 0,Y 377.951,Z 590.72,A -85,B 0,C 180,E1 -12313.249,E2 -12313.249} C_VEL
LIN {X 0,Y 376.773,Z 599.77,A -85,B 0,C 180,E1 -12315.139,E2 -12315.139} C_VEL
LIN {X 0,Y 375.914,Z 607.281,A -85,B 0,C 180,E1 -12317.036,E2 -12317.036} C_VEL
LIN {X 0,Y 375.165,Z 614.29,A -85,B 0,C 180,E1 -12319.203,E2 -12319.203} C_VEL
LIN {X 0,Y 374.785,Z 619.807,A -85,B 0,C 180,E1 -12321.372,E2 -12321.372} C_VEL
LIN {X 0,Y 374.563,Z 623.979,A -85,B 0,C 180,E1 -12323.536,E2 -12323.536} C_VEL
LIN {X 0,Y 374.488,Z 626.905,A -85,B 0,C 180,E1 -12325.695,E2 -12325.695} C_VEL
LIN {X 0,Y 374.452,Z 628.65,A -85,B 0,C 180,E1 -12327.849,E2 -12327.849} C_VEL
LIN {X 0,Y 374.551,Z 629.25,A -85,B 0,C 180,E1 -12330,E2 -12330} C_VEL
LIN {X 0,Y 374.452,Z 628.644,A -85,B 0,C 180,E1 -12332.151,E2 -12332.151} C_VEL
LIN {X 0,Y 374.482,Z 626.891,A -85,B 0,C 180,E1 -12334.305,E2 -12334.305} C_VEL
LIN {X 0,Y 374.562,Z 623.963,A -85,B 0,C 180,E1 -12336.464,E2 -12336.464} C_VEL
LIN {X 0,Y 374.759,Z 619.79,A -85,B 0,C 180,E1 -12338.628,E2 -12338.628} C_VEL
LIN {X 0,Y 375.164,Z 614.265,A -85,B 0,C 180,E1 -12340.797,E2 -12340.797} C_VEL
LIN {X 0,Y 375.911,Z 607.24,A -85,B 0,C 180,E1 -12342.964,E2 -12342.964} C_VEL
LIN {X 0,Y 376.921,Z 598.502,A -85,B 0,C 180,E1 -12345.131,E2 -12345.131} C_VEL
LIN {X 0,Y 378.134,Z 589.225,A -85,B 0,C 180,E1 -12347.021,E2 -12347.021} C_VEL
LIN {X 0,Y 379.568,Z 579.813,A -85,B 0,C 180,E1 -12348.624,E2 -12348.624} C_VEL
LIN {X 0,Y 381.15,Z 567.687,A -85,B 0,C 180,E1 -12350.352,E2 -12350.352} C_VEL
LIN {X 0,Y 382.916,Z 555.124,A -85,B 0,C 180,E1 -12351.818,E2 -12351.818} C_VEL
LIN {X 0,Y 384.457,Z 542.871,A -85,B 0,C 180,E1 -12353,E2 -12353} C_VEL
LIN {X 0,Y 386.161,Z 528.102,A -85,B 0,C 180,E1 -12354.151,E2 -12354.151} C_VEL
LIN {X 0,Y 387.573,Z 513.563,A -85,B 0,C 180,E1 -12355.035,E2 -12355.035} C_VEL
LIN {X 0,Y 388.767,Z 497.768,A -85,B 0,C 180,E1 -12355.748,E2 -12355.748} C_VEL
LIN {X 0,Y 389.626,Z 482.068,A -85,B 0,C 180,E1 -12356.226,E2 -12356.226} C_VEL
LIN {X 0,Y 392.255,Z 370.929,A -85,B 0,C 180,E1 -12358.3,E2 -12358.3} C_VEL
LIN {X 0,Y 392.403,Z 356.593,A -85,B 0,C 180,E1 -12358.58,E2 -12358.58} C_VEL
LIN {X 0,Y 387.82,Z 332.242,A -85,B 0,C 180,E1 -12359.451,E2 -12359.451} C_VEL
LIN {X 0,Y 386.168,Z 325.25,A -85,B 0,C 180,E1 -12359.734,E2 -12359.734} C_VEL
LIN {X 0,Y 382.405,Z 316.48,A -85,B 0,C 180,E1 -12360.256,E2 -12360.256} C_VEL
LIN {X 0,Y 379.448,Z 304.145,A -85,B 0,C 180,E1 -12362.968,E2 -12362.968} C_VEL
LIN {X 0,Y 375.993,Z 291.277,A -85,B 0,C 180,E1 -12365.987,E2 -12365.987} C_VEL
LIN {X 0,Y 375.928,Z 291.284,A -85,B 0,C 180,E1 -12369.466,E2 -12369.466} C_VEL
LIN {X 0,Y 375.927,Z 291.283,A -85,B 0,C 180,E1 -12373.188,E2 -12373.188} C_VEL
LIN {X 0,Y 375.927,Z 291.282,A -85,B 0,C 180,E1 -12376.81,E2 -12376.81} C_VEL
LIN {X 0,Y 375.926,Z 291.283,A -85,B 0,C 180,E1 -12380.533,E2 -12380.533} C_VEL
LIN {X 0,Y 375.948,Z 291.281,A -85,B 0,C 180,E1 -12383.497,E2 -12383.497} C_VEL
LIN {X 0,Y 375.949,Z 291.281,A -85,B 0,C 180,E1 -12385.888,E2 -12385.888} C_VEL
LIN {X 0,Y 375.953,Z 291.277,A -85,B 0,C 180,E1 -12389.686,E2 -12389.686} C_VEL
LIN {X 0,Y 375.917,Z 291.281,A -85,B 0,C 180,E1 -12392.135,E2 -12392.135} C_VEL
LIN {X 0,Y 375.926,Z 291.281,A -85,B 0,C 180,E1 -12394.533,E2 -12394.533} C_VEL
LIN {X 0,Y 375.961,Z 291.275,A -85,B 0,C 180,E1 -12396.886,E2 -12396.886} C_VEL
LIN {X 0,Y 375.985,Z 291.256,A -85,B 0,C 180,E1 -12400.339,E2 -12400.339} C_VEL
LIN {X 0,Y 376.014,Z 291.271,A -85,B 0,C 180,E1 -12403.718,E2 -12403.718} C_VEL
LIN {X 0,Y 376.09,Z 291.248,A -85,B 0,C 180,E1 -12407.042,E2 -12407.042} C_VEL
LIN {X 0,Y 376.094,Z 291.254,A -85,B 0,C 180,E1 -12410.318,E2 -12410.318} C_VEL
LIN {X 0,Y 376.201,Z 291.245,A -85,B 0,C 180,E1 -12413.564,E2 -12413.564} C_VEL
LIN {X 0,Y 376.326,Z 291.227,A -85,B 0,C 180,E1 -12417.86,E2 -12417.86} C_VEL
LIN {X 0,Y 376.33,Z 291.226,A -85,B 0,C 180,E1 -12422.141,E2 -12422.141} C_VEL
LIN {X 0,Y 376.196,Z 291.243,A -85,B 0,C 180,E1 -12426.565,E2 -12426.565} C_VEL
LIN {X 0,Y 376.101,Z 291.258,A -85,B 0,C 180,E1 -12429.682,E2 -12429.682} C_VEL
LIN {X 0,Y 376.08,Z 291.261,A -85,B 0,C 180,E1 -12433.658,E2 -12433.658} C_VEL
LIN {X 0,Y 376.022,Z 291.27,A -85,B 0,C 180,E1 -12437.4,E2 -12437.4} C_VEL
LIN {X 0,Y 375.97,Z 291.254,A -85,B 0,C 180,E1 -12440.833,E2 -12440.833} C_VEL
LIN {X 0,Y 375.973,Z 291.276,A -85,B 0,C 180,E1 -12444.283,E2 -12444.283} C_VEL
LIN {X 0,Y 375.979,Z 291.261,A -85,B 0,C 180,E1 -12446.655,E2 -12446.655} C_VEL
LIN {X 0,Y 375.957,Z 291.278,A -85,B 0,C 180,E1 -12450.313,E2 -12450.313} C_VEL
LIN {X 0,Y 375.95,Z 291.278,A -85,B 0,C 180,E1 -12454.113,E2 -12454.113} C_VEL
LIN {X 0,Y 375.943,Z 291.281,A -85,B 0,C 180,E1 -12456.743,E2 -12456.743} C_VEL
LIN {X 0,Y 375.982,Z 291.271,A -85,B 0,C 180,E1 -12459.971,E2 -12459.971} C_VEL
LIN {X 0,Y 375.924,Z 291.282,A -85,B 0,C 180,E1 -12463.767,E2 -12463.767} C_VEL
LIN {X 0,Y 375.929,Z 291.283,A -85,B 0,C 180,E1 -12466.812,E2 -12466.812} C_VEL
LIN {X 0,Y 375.959,Z 291.274,A -85,B 0,C 180,E1 -12470.538,E2 -12470.538} C_VEL
LIN {X 0,Y 375.96,Z 291.276,A -85,B 0,C 180,E1 -12473.497,E2 -12473.497} C_VEL
LIN {X 0,Y 375.957,Z 291.28,A -85,B 0,C 180,E1 -12475.889,E2 -12475.889} C_VEL
LIN {X 0,Y 375.958,Z 291.39,A -85,B 0,C 180,E1 -12477.641,E2 -12477.641} C_VEL
LIN {X 0,Y 377.826,Z 298.441,A -85,B 0,C 180,E1 -12479.415,E2 -12479.415} C_VEL
LIN {X 0,Y 388.243,Z 320.393,A -85,B 0,C 180,E1 -12480.785,E2 -12480.785} C_VEL
LIN {X 0,Y 393.031,Z 332.171,A -85,B 0,C 180,E1 -12481.419,E2 -12481.419} C_VEL
LIN {X 0,Y 390.502,Z 441.397,A -85,B 0,C 180,E1 -12483.442,E2 -12483.442} C_VEL
LIN {X 0,Y 389.824,Z 465.452,A -85,B 0,C 180,E1 -12483.932,E2 -12483.932} C_VEL
LIN {X 0,Y 389.049,Z 480.629,A -85,B 0,C 180,E1 -12484.447,E2 -12484.447} C_VEL
LIN {X 0,Y 388.155,Z 493.884,A -85,B 0,C 180,E1 -12485.075,E2 -12485.075} C_VEL
LIN {X 0,Y 386.818,Z 508.899,A -85,B 0,C 180,E1 -12486.014,E2 -12486.014} C_VEL
LIN {X 0,Y 385.3,Z 522.149,A -85,B 0,C 180,E1 -12487.053,E2 -12487.053} C_VEL
LIN {X 0,Y 383.652,Z 535.609,A -85,B 0,C 180,E1 -12488.367,E2 -12488.367} C_VEL
LIN {X 0,Y 382.124,Z 546.995,A -85,B 0,C 180,E1 -12489.717,E2 -12489.717} C_VEL
LIN {X 0,Y 380.696,Z 557.168,A -85,B 0,C 180,E1 -12491.152,E2 -12491.152} C_VEL
LIN {X 0,Y 379.305,Z 566.806,A -85,B 0,C 180,E1 -12492.756,E2 -12492.756} C_VEL
LIN {X 0,Y 377.935,Z 576.251,A -85,B 0,C 180,E1 -12494.634,E2 -12494.634} C_VEL
LIN {X 0,Y 376.917,Z 584.108,A -85,B 0,C 180,E1 -12496.522,E2 -12496.522} C_VEL
LIN {X 0,Y 375.913,Z 591.444,A -85,B 0,C 180,E1 -12498.679,E2 -12498.679} C_VEL
LIN {X 0,Y 375.32,Z 597.26,A -85,B 0,C 180,E1 -12500.842,E2 -12500.842} C_VEL
LIN {X 0,Y 374.994,Z 600.703,A -85,B 0,C 180,E1 -12502.462,E2 -12502.462} C_VEL
LIN {X 0,Y 374.74,Z 604.19,A -85,B 0,C 180,E1 -12504.62,E2 -12504.62} C_VEL
LIN {X 0,Y 374.542,Z 606.498,A -85,B 0,C 180,E1 -12506.773,E2 -12506.773} C_VEL
LIN {X 0,Y 374.543,Z 607.674,A -85,B 0,C 180,E1 -12508.925,E2 -12508.925} C_VEL
LIN {X 0,Y 374.543,Z 607.689,A -85,B 0,C 180,E1 -12511.075,E2 -12511.075} C_VEL
LIN {X 0,Y 374.537,Z 606.571,A -85,B 0,C 180,E1 -12513.232,E2 -12513.232} C_VEL
LIN {X 0,Y 374.729,Z 604.327,A -85,B 0,C 180,E1 -12515.381,E2 -12515.381} C_VEL
LIN {X 0,Y 375.02,Z 600.361,A -85,B 0,C 180,E1 -12517.812,E2 -12517.812} C_VEL
LIN {X 0,Y 374.511,Z 598.664,A -85,B 0,C 180,E1 -12518.674,E2 -12518.674} C_VEL
LIN {X 0,Y 371.943,Z 595.656,A -85,B 0,C 180,E1 -12520.073,E2 -12520.073} C_VEL
LIN {X 0,Y 369.526,Z 592.152,A -85,B 0,C 180,E1 -12521.461,E2 -12521.461} C_VEL
LIN {X 0,Y 369.257,Z 589.644,A -85,B 0,C 180,E1 -12522.29,E2 -12522.29} C_VEL
LIN {X 0,Y 370.138,Z 582.633,A -85,B 0,C 180,E1 -12524.29,E2 -12524.29} C_VEL
LIN {X 0,Y 371.378,Z 574.446,A -85,B 0,C 180,E1 -12526.208,E2 -12526.208} C_VEL
LIN {X 0,Y 372.924,Z 564.58,A -85,B 0,C 180,E1 -12528.116,E2 -12528.116} C_VEL
LIN {X 0,Y 374.46,Z 554.463,A -85,B 0,C 180,E1 -12529.744,E2 -12529.744} C_VEL
LIN {X 0,Y 376.008,Z 543.478,A -85,B 0,C 180,E1 -12531.231,E2 -12531.231} C_VEL
LIN {X 0,Y 377.7,Z 531.612,A -85,B 0,C 180,E1 -12532.567,E2 -12532.567} C_VEL
LIN {X 0,Y 379.261,Z 518.767,A -85,B 0,C 180,E1 -12533.768,E2 -12533.768} C_VEL
LIN {X 0,Y 380.78,Z 504.671,A -85,B 0,C 180,E1 -12534.827,E2 -12534.827} C_VEL
LIN {X 0,Y 382.101,Z 489.447,A -85,B 0,C 180,E1 -12535.714,E2 -12535.714} C_VEL
LIN {X 0,Y 383.059,Z 474.781,A -85,B 0,C 180,E1 -12536.344,E2 -12536.344} C_VEL
LIN {X 0,Y 383.771,Z 460.12,A -85,B 0,C 180,E1 -12536.768,E2 -12536.768} C_VEL
LIN {X 0,Y 386.795,Z 335.209,A -85,B 0,C 180,E1 -12539.131,E2 -12539.131} C_VEL
LIN {X 0,Y 386.579,Z 333.07,A -85,B 0,C 180,E1 -12539.193,E2 -12539.193} C_VEL
LIN {X 0,Y 377.471,Z 312.522,A -85,B 0,C 180,E1 -12540.418,E2 -12540.418} C_VEL
LIN {X 0,Y 370.607,Z 298.518,A -85,B 0,C 180,E1 -12541.375,E2 -12541.375} C_VEL
LIN {X 0,Y 368.895,Z 292.165,A -85,B 0,C 180,E1 -12543.042,E2 -12543.042} C_VEL
LIN {X 0,Y 368.915,Z 292.163,A -85,B 0,C 180,E1 -12546.196,E2 -12546.196} C_VEL
LIN {X 0,Y 368.9,Z 292.165,A -85,B 0,C 180,E1 -12548.952,E2 -12548.952} C_VEL
LIN {X 0,Y 368.877,Z 292.163,A -85,B 0,C 180,E1 -12552.008,E2 -12552.008} C_VEL
LIN {X 0,Y 368.874,Z 292.161,A -85,B 0,C 180,E1 -12555.175,E2 -12555.175} C_VEL
LIN {X 0,Y 368.875,Z 292.145,A -85,B 0,C 180,E1 -12558.176,E2 -12558.176} C_VEL
LIN {X 0,Y 368.898,Z 292.156,A -85,B 0,C 180,E1 -12561.36,E2 -12561.36} C_VEL
LIN {X 0,Y 368.924,Z 292.151,A -85,B 0,C 180,E1 -12565.145,E2 -12565.145} C_VEL
LIN {X 0,Y 368.905,Z 292.136,A -85,B 0,C 180,E1 -12569.044,E2 -12569.044} C_VEL
LIN {X 0,Y 368.953,Z 292.15,A -85,B 0,C 180,E1 -12571.562,E2 -12571.562} C_VEL
LIN {X 0,Y 368.936,Z 292.152,A -85,B 0,C 180,E1 -12575.223,E2 -12575.223} C_VEL
LIN {X 0,Y 368.911,Z 292.153,A -85,B 0,C 180,E1 -12578.98,E2 -12578.98} C_VEL
LIN {X 0,Y 368.982,Z 292.141,A -85,B 0,C 180,E1 -12582.257,E2 -12582.257} C_VEL
LIN {X 0,Y 369.028,Z 292.137,A -85,B 0,C 180,E1 -12586.228,E2 -12586.228} C_VEL
LIN {X 0,Y 369.052,Z 292.136,A -85,B 0,C 180,E1 -12590.131,E2 -12590.131} C_VEL
LIN {X 0,Y 369.168,Z 292.123,A -85,B 0,C 180,E1 -12593.441,E2 -12593.441} C_VEL
LIN {X 0,Y 369.297,Z 292.107,A -85,B 0,C 180,E1 -12597.819,E2 -12597.819} C_VEL
LIN {X 0,Y 369.42,Z 292.086,A -85,B 0,C 180,E1 -12600,E2 -12600} C_VEL
LIN {X 0,Y 369.291,Z 292.108,A -85,B 0,C 180,E1 -12602.181,E2 -12602.181} C_VEL
LIN {X 0,Y 369.167,Z 292.127,A -85,B 0,C 180,E1 -12606.559,E2 -12606.559} C_VEL
LIN {X 0,Y 369.049,Z 292.133,A -85,B 0,C 180,E1 -12609.869,E2 -12609.869} C_VEL
LIN {X 0,Y 369.027,Z 292.134,A -85,B 0,C 180,E1 -12613.772,E2 -12613.772} C_VEL
LIN {X 0,Y 368.981,Z 292.143,A -85,B 0,C 180,E1 -12617.743,E2 -12617.743} C_VEL
LIN {X 0,Y 368.899,Z 292.155,A -85,B 0,C 180,E1 -12621.221,E2 -12621.221} C_VEL
LIN {X 0,Y 368.906,Z 292.159,A -85,B 0,C 180,E1 -12623.877,E2 -12623.877} C_VEL
LIN {X 0,Y 368.859,Z 292.162,A -85,B 0,C 180,E1 -12627.212,E2 -12627.212} C_VEL
LIN {X 0,Y 368.886,Z 292.16,A -85,B 0,C 180,E1 -12629.693,E2 -12629.693} C_VEL
LIN {X 0,Y 368.888,Z 292.151,A -85,B 0,C 180,E1 -12633.043,E2 -12633.043} C_VEL
LIN {X 0,Y 368.902,Z 292.154,A -85,B 0,C 180,E1 -12636.198,E2 -12636.198} C_VEL
LIN {X 0,Y 368.865,Z 292.157,A -85,B 0,C 180,E1 -12638.958,E2 -12638.958} C_VEL
LIN {X 0,Y 368.863,Z 292.154,A -85,B 0,C 180,E1 -12642.008,E2 -12642.008} C_VEL
LIN {X 0,Y 368.868,Z 292.162,A -85,B 0,C 180,E1 -12645.176,E2 -12645.176} C_VEL
LIN {X 0,Y 368.854,Z 292.162,A -85,B 0,C 180,E1 -12648.175,E2 -12648.175} C_VEL
LIN {X 0,Y 368.87,Z 292.16,A -85,B 0,C 180,E1 -12651.367,E2 -12651.367} C_VEL
LIN {X 0,Y 368.934,Z 292.262,A -85,B 0,C 180,E1 -12653.479,E2 -12653.479} C_VEL
LIN {X 0,Y 372.398,Z 304.889,A -85,B 0,C 180,E1 -12656.509,E2 -12656.509} C_VEL
LIN {X 0,Y 375.199,Z 316.47,A -85,B 0,C 180,E1 -12659.105,E2 -12659.105} C_VEL
LIN {X 0,Y 380.997,Z 330.003,A -85,B 0,C 180,E1 -12659.911,E2 -12659.911} C_VEL
LIN {X 0,Y 386.228,Z 357.668,A -85,B 0,C 180,E1 -12660.933,E2 -12660.933} C_VEL
LIN {X 0,Y 384.343,Z 442.524,A -85,B 0,C 180,E1 -12662.54,E2 -12662.54} C_VEL
LIN {X 0,Y 383.251,Z 483.647,A -85,B 0,C 180,E1 -12663.34,E2 -12663.34} C_VEL
LIN {X 0,Y 382.375,Z 498.702,A -85,B 0,C 180,E1 -12663.826,E2 -12663.826} C_VEL
LIN {X 0,Y 381.117,Z 513.762,A -85,B 0,C 180,E1 -12664.524,E2 -12664.524} C_VEL
LIN {X 0,Y 379.626,Z 528.512,A -85,B 0,C 180,E1 -12665.442,E2 -12665.442} C_VEL
LIN {X 0,Y 377.872,Z 542.783,A -85,B 0,C 180,E1 -12666.576,E2 -12666.576} C_VEL
LIN {X 0,Y 376.05,Z 556.225,A -85,B 0,C 180,E1 -12667.907,E2 -12667.907} C_VEL
LIN {X 0,Y 374.289,Z 568.471,A -85,B 0,C 180,E1 -12669.387,E2 -12669.387} C_VEL
LIN {X 0,Y 372.746,Z 579.852,A -85,B 0,C 180,E1 -12671.053,E2 -12671.053} C_VEL
LIN {X 0,Y 371.068,Z 590.517,A -85,B 0,C 180,E1 -12672.929,E2 -12672.929} C_VEL
LIN {X 0,Y 369.83,Z 599.566,A -85,B 0,C 180,E1 -12674.853,E2 -12674.853} C_VEL
LIN {X 0,Y 368.919,Z 607.077,A -85,B 0,C 180,E1 -12676.786,E2 -12676.786} C_VEL
LIN {X 0,Y 368.148,Z 614.087,A -85,B 0,C 180,E1 -12678.995,E2 -12678.995} C_VEL
LIN {X 0,Y 367.721,Z 619.604,A -85,B 0,C 180,E1 -12681.205,E2 -12681.205} C_VEL
LIN {X 0,Y 367.481,Z 623.776,A -85,B 0,C 180,E1 -12683.411,E2 -12683.411} C_VEL
LIN {X 0,Y 367.397,Z 626.702,A -85,B 0,C 180,E1 -12685.612,E2 -12685.612} C_VEL
LIN {X 0,Y 367.352,Z 628.447,A -85,B 0,C 180,E1 -12687.807,E2 -12687.807} C_VEL
LIN {X 0,Y 367.454,Z 629.047,A -85,B 0,C 180,E1 -12690,E2 -12690} C_VEL
LIN {X 0,Y 367.352,Z 628.441,A -85,B 0,C 180,E1 -12692.193,E2 -12692.193} C_VEL
LIN {X 0,Y 367.39,Z 626.688,A -85,B 0,C 180,E1 -12694.388,E2 -12694.388} C_VEL
LIN {X 0,Y 367.479,Z 623.758,A -85,B 0,C 180,E1 -12696.589,E2 -12696.589} C_VEL
LIN {X 0,Y 367.704,Z 619.585,A -85,B 0,C 180,E1 -12698.795,E2 -12698.795} C_VEL
LIN {X 0,Y 368.147,Z 614.059,A -85,B 0,C 180,E1 -12701.005,E2 -12701.005} C_VEL
LIN {X 0,Y 368.909,Z 607.033,A -85,B 0,C 180,E1 -12703.215,E2 -12703.215} C_VEL
LIN {X 0,Y 369.997,Z 598.296,A -85,B 0,C 180,E1 -12705.422,E2 -12705.422} C_VEL
LIN {X 0,Y 371.267,Z 589.018,A -85,B 0,C 180,E1 -12707.346,E2 -12707.346} C_VEL
LIN {X 0,Y 372.757,Z 579.766,A -85,B 0,C 180,E1 -12708.95,E2 -12708.95} C_VEL
LIN {X 0,Y 374.265,Z 568.593,A -85,B 0,C 180,E1 -12710.586,E2 -12710.586} C_VEL
LIN {X 0,Y 376.116,Z 556.14,A -85,B 0,C 180,E1 -12712.089,E2 -12712.089} C_VEL
LIN {X 0,Y 377.914,Z 542.663,A -85,B 0,C 180,E1 -12713.422,E2 -12713.422} C_VEL
LIN {X 0,Y 379.626,Z 528.373,A -85,B 0,C 180,E1 -12714.557,E2 -12714.557} C_VEL
LIN {X 0,Y 381.111,Z 513.352,A -85,B 0,C 180,E1 -12715.49,E2 -12715.49} C_VEL
LIN {X 0,Y 382.402,Z 497.555,A -85,B 0,C 180,E1 -12716.209,E2 -12716.209} C_VEL
LIN {X 0,Y 383.256,Z 481.848,A -85,B 0,C 180,E1 -12716.696,E2 -12716.696} C_VEL
LIN {X 0,Y 385.668,Z 384.204,A -85,B 0,C 180,E1 -12718.547,E2 -12718.547} C_VEL
LIN {X 0,Y 386.168,Z 357.688,A -85,B 0,C 180,E1 -12719.057,E2 -12719.057} C_VEL
LIN {X 0,Y 380.949,Z 330.081,A -85,B 0,C 180,E1 -12720.077,E2 -12720.077} C_VEL
LIN {X 0,Y 378.317,Z 323.464,A -85,B 0,C 180,E1 -12720.448,E2 -12720.448} C_VEL
LIN {X 0,Y 375.158,Z 316.33,A -85,B 0,C 180,E1 -12720.886,E2 -12720.886} C_VEL
LIN {X 0,Y 372.031,Z 303.585,A -85,B 0,C 180,E1 -12723.778,E2 -12723.778} C_VEL
LIN {X 0,Y 368.923,Z 292.155,A -85,B 0,C 180,E1 -12726.547,E2 -12726.547} C_VEL
LIN {X 0,Y 368.878,Z 292.166,A -85,B 0,C 180,E1 -12730.373,E2 -12730.373} C_VEL
LIN {X 0,Y 368.874,Z 292.162,A -85,B 0,C 180,E1 -12733.615,E2 -12733.615} C_VEL
LIN {X 0,Y 368.878,Z 292.161,A -85,B 0,C 180,E1 -12736.695,E2 -12736.695} C_VEL
LIN {X 0,Y 368.877,Z 292.16,A -85,B 0,C 180,E1 -12739.648,E2 -12739.648} C_VEL
LIN {X 0,Y 368.887,Z 292.158,A -85,B 0,C 180,E1 -12743.145,E2 -12743.145} C_VEL
LIN {X 0,Y 368.887,Z 292.156,A -85,B 0,C 180,E1 -12746.461,E2 -12746.461} C_VEL
LIN {X 0,Y 368.904,Z 292.156,A -85,B 0,C 180,E1 -12749.044,E2 -12749.044} C_VEL
LIN {X 0,Y 368.902,Z 292.159,A -85,B 0,C 180,E1 -12751.558,E2 -12751.558} C_VEL
LIN {X 0,Y 368.876,Z 292.161,A -85,B 0,C 180,E1 -12755.219,E2 -12755.219} C_VEL
LIN {X 0,Y 368.908,Z 292.159,A -85,B 0,C 180,E1 -12757.603,E2 -12757.603} C_VEL
LIN {X 0,Y 368.943,Z 292.13,A -85,B 0,C 180,E1 -12761.105,E2 -12761.105} C_VEL
LIN {X 0,Y 368.985,Z 292.146,A -85,B 0,C 180,E1 -12764.535,E2 -12764.535} C_VEL
LIN {X 0,Y 369.046,Z 292.13,A -85,B 0,C 180,E1 -12766.79,E2 -12766.79} C_VEL
LIN {X 0,Y 369.045,Z 292.128,A -85,B 0,C 180,E1 -12770.131,E2 -12770.131} C_VEL
LIN {X 0,Y 369.161,Z 292.123,A -85,B 0,C 180,E1 -12773.441,E2 -12773.441} C_VEL
LIN {X 0,Y 369.29,Z 292.103,A -85,B 0,C 180,E1 -12777.819,E2 -12777.819} C_VEL
LIN {X 0,Y 369.294,Z 292.102,A -85,B 0,C 180,E1 -12782.181,E2 -12782.181} C_VEL
LIN {X 0,Y 369.168,Z 292.119,A -85,B 0,C 180,E1 -12786.559,E2 -12786.559} C_VEL
LIN {X 0,Y 369.052,Z 292.135,A -85,B 0,C 180,E1 -12789.869,E2 -12789.869} C_VEL
LIN {X 0,Y 369.028,Z 292.139,A -85,B 0,C 180,E1 -12793.772,E2 -12793.772} C_VEL
LIN {X 0,Y 368.982,Z 292.144,A -85,B 0,C 180,E1 -12797.743,E2 -12797.743} C_VEL
LIN {X 0,Y 368.901,Z 292.136,A -85,B 0,C 180,E1 -12801.222,E2 -12801.222} C_VEL
LIN {X 0,Y 368.937,Z 292.155,A -85,B 0,C 180,E1 -12804.777,E2 -12804.777} C_VEL
LIN {X 0,Y 368.954,Z 292.136,A -85,B 0,C 180,E1 -12808.438,E2 -12808.438} C_VEL
LIN {X 0,Y 368.889,Z 292.154,A -85,B 0,C 180,E1 -12812.239,E2 -12812.239} C_VEL
LIN {X 0,Y 368.916,Z 292.154,A -85,B 0,C 180,E1 -12815.001,E2 -12815.001} C_VEL
LIN {X 0,Y 368.901,Z 292.157,A -85,B 0,C 180,E1 -12818.641,E2 -12818.641} C_VEL
LIN {X 0,Y 368.875,Z 292.159,A -85,B 0,C 180,E1 -12822.01,E2 -12822.01} C_VEL
LIN {X 0,Y 368.875,Z 292.162,A -85,B 0,C 180,E1 -12825.177,E2 -12825.177} C_VEL
LIN {X 0,Y 368.879,Z 292.163,A -85,B 0,C 180,E1 -12828.178,E2 -12828.178} C_VEL
LIN {X 0,Y 368.905,Z 292.149,A -85,B 0,C 180,E1 -12831.361,E2 -12831.361} C_VEL
LIN {X 0,Y 368.933,Z 292.153,A -85,B 0,C 180,E1 -12835.147,E2 -12835.147} C_VEL
LIN {X 0,Y 368.924,Z 292.249,A -85,B 0,C 180,E1 -12837.097,E2 -12837.097} C_VEL
LIN {X 0,Y 370.596,Z 298.628,A -85,B 0,C 180,E1 -12838.75,E2 -12838.75} C_VEL
LIN {X 0,Y 381.658,Z 321.587,A -85,B 0,C 180,E1 -12840.251,E2 -12840.251} C_VEL
LIN {X 0,Y 386.739,Z 333.624,A -85,B 0,C 180,E1 -12840.936,E2 -12840.936} C_VEL
LIN {X 0,Y 384.236,Z 439.837,A -85,B 0,C 180,E1 -12842.937,E2 -12842.937} C_VEL
LIN {X 0,Y 383.51,Z 464.532,A -85,B 0,C 180,E1 -12843.433,E2 -12843.433} C_VEL
LIN {X 0,Y 382.755,Z 479.98,A -85,B 0,C 180,E1 -12843.955,E2 -12843.955} C_VEL
LIN {X 0,Y 381.693,Z 494.684,A -85,B 0,C 180,E1 -12844.662,E2 -12844.662} C_VEL
LIN {X 0,Y 380.346,Z 509.108,A -85,B 0,C 180,E1 -12845.579,E2 -12845.579} C_VEL
LIN {X 0,Y 378.764,Z 522.358,A -85,B 0,C 180,E1 -12846.634,E2 -12846.634} C_VEL
LIN {X 0,Y 377.066,Z 535.816,A -85,B 0,C 180,E1 -12847.97,E2 -12847.97} C_VEL
LIN {X 0,Y 375.352,Z 547.839,A -85,B 0,C 180,E1 -12849.421,E2 -12849.421} C_VEL
LIN {X 0,Y 373.704,Z 559.142,A -85,B 0,C 180,E1 -12851.071,E2 -12851.071} C_VEL
LIN {X 0,Y 372.082,Z 569.937,A -85,B 0,C 180,E1 -12852.977,E2 -12852.977} C_VEL
LIN {X 0,Y 370.692,Z 579.011,A -85,B 0,C 180,E1 -12854.918,E2 -12854.918} C_VEL
LIN {X 0,Y 369.73,Z 586.312,A -85,B 0,C 180,E1 -12856.815,E2 -12856.815} C_VEL
LIN {X 0,Y 368.736,Z 593.248,A -85,B 0,C 180,E1 -12859.013,E2 -12859.013} C_VEL
LIN {X 0,Y 368.176,Z 598.692,A -85,B 0,C 180,E1 -12861.216,E2 -12861.216} C_VEL
LIN {X 0,Y 367.785,Z 603.016,A -85,B 0,C 180,E1 -12863.55,E2 -12863.55} C_VEL
LIN {X 0,Y 367.552,Z 605.691,A -85,B 0,C 180,E1 -12865.614,E2 -12865.614} C_VEL
LIN {X 0,Y 367.444,Z 607.428,A -85,B 0,C 180,E1 -12867.808,E2 -12867.808} C_VEL
LIN {X 0,Y 367.456,Z 608.034,A -85,B 0,C 180,E1 -12870,E2 -12870} C_VEL
LIN {X 0,Y 367.443,Z 607.474,A -85,B 0,C 180,E1 -12872.192,E2 -12872.192} C_VEL
LIN {X 0,Y 367.545,Z 605.797,A -85,B 0,C 180,E1 -12874.386,E2 -12874.386} C_VEL
LIN {X 0,Y 367.764,Z 602.966,A -85,B 0,C 180,E1 -12876.584,E2 -12876.584} C_VEL
LIN {X 0,Y 368.141,Z 598.912,A -85,B 0,C 180,E1 -12878.785,E2 -12878.785} C_VEL
LIN {X 0,Y 368.709,Z 593.537,A -85,B 0,C 180,E1 -12880.988,E2 -12880.988} C_VEL
LIN {X 0,Y 369.257,Z 589.644,A -85,B 0,C 180,E1 -12882.29,E2 -12882.29} C_VEL
LIN {X 0,Y 369.021,Z 587.049,A -85,B 0,C 180,E1 -12883.11,E2 -12883.11} C_VEL
LIN {X 0,Y 366.821,Z 582.667,A -85,B 0,C 180,E1 -12884.459,E2 -12884.459} C_VEL
LIN {X 0,Y 364.695,Z 577.872,A -85,B 0,C 180,E1 -12885.781,E2 -12885.781} C_VEL
LIN {X 0,Y 364.568,Z 574.52,A -85,B 0,C 180,E1 -12886.547,E2 -12886.547} C_VEL
LIN {X 0,Y 366.14,Z 564.782,A -85,B 0,C 180,E1 -12888.464,E2 -12888.464} C_VEL
LIN {X 0,Y 367.953,Z 553.254,A -85,B 0,C 180,E1 -12890.331,E2 -12890.331} C_VEL
LIN {X 0,Y 369.678,Z 541.51,A -85,B 0,C 180,E1 -12891.906,E2 -12891.906} C_VEL
LIN {X 0,Y 371.487,Z 529.232,A -85,B 0,C 180,E1 -12893.261,E2 -12893.261} C_VEL
LIN {X 0,Y 373.191,Z 515.808,A -85,B 0,C 180,E1 -12894.475,E2 -12894.475} C_VEL
